LIN {X 0,Y 207.071,Z 348.497,A -85,B 0,C 180,E1 -23061.924,E2 -23061.924} C_VEL
LIN {X 0,Y 208.464,Z 354.265,A -85,B 0,C 180,E1 -23067.075,E2 -23067.075} C_VEL
LIN {X 0,Y 209.704,Z 358.969,A -85,B 0,C 180,E1 -23070.181,E2 -23070.181} C_VEL
LIN {X 0,Y 211.466,Z 367.193,A -85,B 0,C 180,E1 -23074.403,E2 -23074.403} C_VEL
LIN {X 0,Y 212.474,Z 373.609,A -85,B 0,C 180,E1 -23077.134,E2 -23077.134} C_VEL
LIN {X 0,Y 211.976,Z 381.158,A -85,B 0,C 180,E1 -23079.446,E2 -23079.446} C_VEL
LIN {X 0,Y 210.448,Z 390.937,A -85,B 0,C 180,E1 -23082.249,E2 -23082.249} C_VEL
LIN {X 0,Y 208.137,Z 400.366,A -85,B 0,C 180,E1 -23084.841,E2 -23084.841} C_VEL
LIN {X 0,Y 206.322,Z 405.58,A -85,B 0,C 180,E1 -23086.272,E2 -23086.272} C_VEL
LIN {X 0,Y 199.113,Z 417.683,A -85,B 0,C 180,E1 -23089.235,E2 -23089.235} C_VEL
LIN {X 0,Y 192.772,Z 427.559,A -85,B 0,C 180,E1 -23092.364,E2 -23092.364} C_VEL
LIN {X 0,Y 186.872,Z 436.167,A -85,B 0,C 180,E1 -23095.835,E2 -23095.835} C_VEL
LIN {X 0,Y 181.675,Z 443.782,A -85,B 0,C 180,E1 -23099.81,E2 -23099.81} C_VEL
LIN {X 0,Y 177.015,Z 450.226,A -85,B 0,C 180,E1 -23104.106,E2 -23104.106} C_VEL
LIN {X 0,Y 173.093,Z 455.772,A -85,B 0,C 180,E1 -23109.049,E2 -23109.049} C_VEL
LIN {X 0,Y 171.048,Z 459.248,A -85,B 0,C 180,E1 -23113.286,E2 -23113.286} C_VEL
LIN {X 0,Y 169.61,Z 461.995,A -85,B 0,C 180,E1 -23118.045,E2 -23118.045} C_VEL
LIN {X 0,Y 169.147,Z 463.562,A -85,B 0,C 180,E1 -23122.841,E2 -23122.841} C_VEL
LIN {X 0,Y 169.224,Z 463.943,A -85,B 0,C 180,E1 -23125.393,E2 -23125.393} C_VEL
LIN {X 0,Y 169.399,Z 463.779,A -85,B 0,C 180,E1 -23129.986,E2 -23129.986} C_VEL
LIN {X 0,Y 169.181,Z 463.569,A -85,B 0,C 180,E1 -23131.308,E2 -23131.308} C_VEL
LIN {X 0,Y 168.389,Z 463.209,A -85,B 0,C 180,E1 -23132.61,E2 -23132.61} C_VEL
LIN {X 0,Y 165.89,Z 462.118,A -85,B 0,C 180,E1 -23135.171,E2 -23135.171} C_VEL
LIN {X 0,Y 163.361,Z 460.595,A -85,B 0,C 180,E1 -23137.794,E2 -23137.794} C_VEL
LIN {X 0,Y 162.39,Z 459.234,A -85,B 0,C 180,E1 -23139.828,E2 -23139.828} C_VEL
LIN {X 0,Y 162.378,Z 458.73,A -85,B 0,C 180,E1 -23140.514,E2 -23140.514} C_VEL
LIN {X 0,Y 163.318,Z 455.126,A -85,B 0,C 180,E1 -23144.965,E2 -23144.965} C_VEL
LIN {X 0,Y 165.316,Z 449.724,A -85,B 0,C 180,E1 -23149.885,E2 -23149.885} C_VEL
LIN {X 0,Y 168.323,Z 442.8,A -85,B 0,C 180,E1 -23154.68,E2 -23154.68} C_VEL
LIN {X 0,Y 172.5,Z 434.174,A -85,B 0,C 180,E1 -23159.27,E2 -23159.27} C_VEL
LIN {X 0,Y 176.98,Z 424.366,A -85,B 0,C 180,E1 -23163.357,E2 -23163.357} C_VEL
LIN {X 0,Y 182.008,Z 413.854,A -85,B 0,C 180,E1 -23166.765,E2 -23166.765} C_VEL
LIN {X 0,Y 186.944,Z 402.449,A -85,B 0,C 180,E1 -23169.727,E2 -23169.727} C_VEL
LIN {X 0,Y 189.021,Z 397.038,A -85,B 0,C 180,E1 -23170.945,E2 -23170.945} C_VEL
LIN {X 0,Y 189.629,Z 386.332,A -85,B 0,C 180,E1 -23173.653,E2 -23173.653} C_VEL
LIN {X 0,Y 189.573,Z 374.931,A -85,B 0,C 180,E1 -23176.331,E2 -23176.331} C_VEL
LIN {X 0,Y 188.758,Z 362.703,A -85,B 0,C 180,E1 -23179.056,E2 -23179.056} C_VEL
LIN {X 0,Y 187.425,Z 353.021,A -85,B 0,C 180,E1 -23181.158,E2 -23181.158} C_VEL
LIN {X 0,Y 185.608,Z 346.725,A -85,B 0,C 180,E1 -23182.709,E2 -23182.709} C_VEL
LIN {X 0,Y 181.291,Z 336.124,A -85,B 0,C 180,E1 -23185.628,E2 -23185.628} C_VEL
LIN {X 0,Y 177.317,Z 327.465,A -85,B 0,C 180,E1 -23188.151,E2 -23188.151} C_VEL
LIN {X 0,Y 174.427,Z 321.833,A -85,B 0,C 180,E1 -23189.923,E2 -23189.923} C_VEL
LIN {X 0,Y 171.849,Z 316.911,A -85,B 0,C 180,E1 -23191.528,E2 -23191.528} C_VEL
LIN {X 0,Y 169.571,Z 313.23,A -85,B 0,C 180,E1 -23192.874,E2 -23192.874} C_VEL
LIN {X 0,Y 168.653,Z 311.253,A -85,B 0,C 180,E1 -23193.468,E2 -23193.468} C_VEL
LIN {X 0,Y 166.254,Z 308.021,A -85,B 0,C 180,E1 -23194.898,E2 -23194.898} C_VEL
LIN {X 0,Y 165.335,Z 305.195,A -85,B 0,C 180,E1 -23195.68,E2 -23195.68} C_VEL
LIN {X 0,Y 165.069,Z 302.898,A -85,B 0,C 180,E1 -23200.083,E2 -23200.083} C_VEL
LIN {X 0,Y 164.708,Z 300.494,A -85,B 0,C 180,E1 -23205.164,E2 -23205.164} C_VEL
LIN {X 0,Y 164.624,Z 299.609,A -85,B 0,C 180,E1 -23207.673,E2 -23207.673} C_VEL
LIN {X 0,Y 164.832,Z 299.582,A -85,B 0,C 180,E1 -23212.649,E2 -23212.649} C_VEL
LIN {X 0,Y 165.05,Z 299.552,A -85,B 0,C 180,E1 -23217.557,E2 -23217.557} C_VEL
LIN {X 0,Y 165.3,Z 299.52,A -85,B 0,C 180,E1 -23219.997,E2 -23219.997} C_VEL
LIN {X 0,Y 164.865,Z 299.571,A -85,B 0,C 180,E1 -23227.345,E2 -23227.345} C_VEL
LIN {X 0,Y 164.752,Z 299.566,A -85,B 0,C 180,E1 -23231.14,E2 -23231.14} C_VEL
LIN {X 0,Y 164.487,Z 299.615,A -85,B 0,C 180,E1 -23237.4,E2 -23237.4} C_VEL
LIN {X 0,Y 164.476,Z 299.597,A -85,B 0,C 180,E1 -23239.986,E2 -23239.986} C_VEL
LIN {X 0,Y 164.394,Z 299.621,A -85,B 0,C 180,E1 -23246.13,E2 -23246.13} C_VEL
LIN {X 0,Y 164.374,Z 299.633,A -85,B 0,C 180,E1 -23251.224,E2 -23251.224} C_VEL
LIN {X 0,Y 164.311,Z 299.623,A -85,B 0,C 180,E1 -23256.781,E2 -23256.781} C_VEL
LIN {X 0,Y 164.302,Z 299.643,A -85,B 0,C 180,E1 -23259.909,E2 -23259.909} C_VEL
LIN {X 0,Y 164.304,Z 299.623,A -85,B 0,C 180,E1 -23263.349,E2 -23263.349} C_VEL
LIN {X 0,Y 164.354,Z 299.637,A -85,B 0,C 180,E1 -23266.827,E2 -23266.827} C_VEL
LIN {X 0,Y 164.367,Z 299.621,A -85,B 0,C 180,E1 -23270.317,E2 -23270.317} C_VEL
LIN {X 0,Y 164.34,Z 299.626,A -85,B 0,C 180,E1 -23274.339,E2 -23274.339} C_VEL
LIN {X 0,Y 164.38,Z 299.747,A -85,B 0,C 180,E1 -23277.96,E2 -23277.96} C_VEL
LIN {X 0,Y 165.251,Z 302.251,A -85,B 0,C 180,E1 -23278.667,E2 -23278.667} C_VEL
LIN {X 0,Y 167.493,Z 304.644,A -85,B 0,C 180,E1 -23280.056,E2 -23280.056} C_VEL
LIN {X 0,Y 168.139,Z 305.575,A -85,B 0,C 180,E1 -23280.472,E2 -23280.472} C_VEL
LIN {X 0,Y 170.033,Z 308.606,A -85,B 0,C 180,E1 -23281.701,E2 -23281.701} C_VEL
LIN {X 0,Y 171.417,Z 310.257,A -85,B 0,C 180,E1 -23282.532,E2 -23282.532} C_VEL
LIN {X 0,Y 173.819,Z 313.919,A -85,B 0,C 180,E1 -23284.055,E2 -23284.055} C_VEL
LIN {X 0,Y 179.648,Z 323.432,A -85,B 0,C 180,E1 -23287.675,E2 -23287.675} C_VEL
LIN {X 0,Y 184.401,Z 332.346,A -85,B 0,C 180,E1 -23290.779,E2 -23290.779} C_VEL
LIN {X 0,Y 189.654,Z 343.67,A -85,B 0,C 180,E1 -23294.456,E2 -23294.456} C_VEL
LIN {X 0,Y 191.768,Z 349.873,A -85,B 0,C 180,E1 -23296.3,E2 -23296.3} C_VEL
LIN {X 0,Y 193.343,Z 355.545,A -85,B 0,C 180,E1 -23297.935,E2 -23297.935} C_VEL
LIN {X 0,Y 194.691,Z 366.513,A -85,B 0,C 180,E1 -23300.886,E2 -23300.886} C_VEL
LIN {X 0,Y 190.147,Z 378.986,A -85,B 0,C 180,E1 -23303.337,E2 -23303.337} C_VEL
LIN {X 0,Y 185.373,Z 390.665,A -85,B 0,C 180,E1 -23306.194,E2 -23306.194} C_VEL
LIN {X 0,Y 180.718,Z 401.146,A -85,B 0,C 180,E1 -23309.386,E2 -23309.386} C_VEL
LIN {X 0,Y 175.962,Z 411.116,A -85,B 0,C 180,E1 -23313.188,E2 -23313.188} C_VEL
LIN {X 0,Y 172.035,Z 419.15,A -85,B 0,C 180,E1 -23317.038,E2 -23317.038} C_VEL
LIN {X 0,Y 169.033,Z 425.451,A -85,B 0,C 180,E1 -23320.782,E2 -23320.782} C_VEL
LIN {X 0,Y 166.504,Z 430.703,A -85,B 0,C 180,E1 -23324.668,E2 -23324.668} C_VEL
LIN {X 0,Y 164.218,Z 435.982,A -85,B 0,C 180,E1 -23329.7,E2 -23329.7} C_VEL
LIN {X 0,Y 162.694,Z 439.901,A -85,B 0,C 180,E1 -23334.893,E2 -23334.893} C_VEL
LIN {X 0,Y 161.98,Z 442.359,A -85,B 0,C 180,E1 -23339.807,E2 -23339.807} C_VEL
LIN {X 0,Y 161.931,Z 443.673,A -85,B 0,C 180,E1 -23344.456,E2 -23344.456} C_VEL
LIN {X 0,Y 162.435,Z 443.957,A -85,B 0,C 180,E1 -23348.855,E2 -23348.855} C_VEL
LIN {X 0,Y 163.587,Z 443.389,A -85,B 0,C 180,E1 -23353.421,E2 -23353.421} C_VEL
LIN {X 0,Y 165.021,Z 442.215,A -85,B 0,C 180,E1 -23357.05,E2 -23357.05} C_VEL
LIN {X 0,Y 168.232,Z 439.191,A -85,B 0,C 180,E1 -23362.533,E2 -23362.533} C_VEL
LIN {X 0,Y 171.634,Z 435.639,A -85,B 0,C 180,E1 -23366.811,E2 -23366.811} C_VEL
LIN {X 0,Y 176.458,Z 430.293,A -85,B 0,C 180,E1 -23371.452,E2 -23371.452} C_VEL
LIN {X 0,Y 181.905,Z 423.855,A -85,B 0,C 180,E1 -23375.596,E2 -23375.596} C_VEL
LIN {X 0,Y 187.841,Z 416.383,A -85,B 0,C 180,E1 -23379.282,E2 -23379.282} C_VEL
LIN {X 0,Y 194.656,Z 407.022,A -85,B 0,C 180,E1 -23382.818,E2 -23382.818} C_VEL
LIN {X 0,Y 201.597,Z 396.484,A -85,B 0,C 180,E1 -23385.878,E2 -23385.878} C_VEL
LIN {X 0,Y 208.063,Z 385.523,A -85,B 0,C 180,E1 -23388.391,E2 -23388.391} C_VEL
LIN {X 0,Y 209.506,Z 382.789,A -85,B 0,C 180,E1 -23388.942,E2 -23388.942} C_VEL
LIN {X 0,Y 210.087,Z 381.064,A -85,B 0,C 180,E1 -23389.44,E2 -23389.44} C_VEL
LIN {X 0,Y 210.237,Z 375.206,A -85,B 0,C 180,E1 -23391.834,E2 -23391.834} C_VEL
LIN {X 0,Y 209.861,Z 370.028,A -85,B 0,C 180,E1 -23394.236,E2 -23394.236} C_VEL
LIN {X 0,Y 208.905,Z 364.791,A -85,B 0,C 180,E1 -23397.11,E2 -23397.11} C_VEL
LIN {X 0,Y 207.74,Z 360.431,A -85,B 0,C 180,E1 -23400.002,E2 -23400.002} C_VEL
LIN {X 0,Y 206.324,Z 355.745,A -85,B 0,C 180,E1 -23403.908,E2 -23403.908} C_VEL
LIN {X 0,Y 204.735,Z 353.325,A -85,B 0,C 180,E1 -23407.894,E2 -23407.894} C_VEL
LIN {X 0,Y 204.53,Z 351.869,A -85,B 0,C 180,E1 -23409.895,E2 -23409.895} C_VEL
LIN {X 0,Y 203.403,Z 352.092,A -85,B 0,C 180,E1 -23414.663,E2 -23414.663} C_VEL
LIN {X 0,Y 203.38,Z 353.038,A -85,B 0,C 180,E1 -23418.122,E2 -23418.122} C_VEL
LIN {X 0,Y 203.937,Z 354.716,A -85,B 0,C 180,E1 -23421.497,E2 -23421.497} C_VEL
LIN {X 0,Y 205.005,Z 360.752,A -85,B 0,C 180,E1 -23426.962,E2 -23426.962} C_VEL
LIN {X 0,Y 205.992,Z 365.65,A -85,B 0,C 180,E1 -23430.2,E2 -23430.2} C_VEL
LIN {X 0,Y 207.088,Z 372.068,A -85,B 0,C 180,E1 -23433.654,E2 -23433.654} C_VEL
LIN {X 0,Y 207.745,Z 377.925,A -85,B 0,C 180,E1 -23436.302,E2 -23436.302} C_VEL
LIN {X 0,Y 206.849,Z 385.122,A -85,B 0,C 180,E1 -23438.608,E2 -23438.608} C_VEL
LIN {X 0,Y 205.232,Z 393.476,A -85,B 0,C 180,E1 -23441.119,E2 -23441.119} C_VEL
LIN {X 0,Y 202.32,Z 403.303,A -85,B 0,C 180,E1 -23444.009,E2 -23444.009} C_VEL
LIN {X 0,Y 200.971,Z 406.814,A -85,B 0,C 180,E1 -23445.002,E2 -23445.002} C_VEL
LIN {X 0,Y 193.8,Z 418.149,A -85,B 0,C 180,E1 -23447.867,E2 -23447.867} C_VEL
LIN {X 0,Y 187.193,Z 427.848,A -85,B 0,C 180,E1 -23451.036,E2 -23451.036} C_VEL
LIN {X 0,Y 180.722,Z 436.732,A -85,B 0,C 180,E1 -23454.755,E2 -23454.755} C_VEL
LIN {X 0,Y 175.535,Z 443.838,A -85,B 0,C 180,E1 -23458.637,E2 -23458.637} C_VEL
LIN {X 0,Y 170.589,Z 450.155,A -85,B 0,C 180,E1 -23463.054,E2 -23463.054} C_VEL
LIN {X 0,Y 166.237,Z 455.858,A -85,B 0,C 180,E1 -23468.454,E2 -23468.454} C_VEL
LIN {X 0,Y 164.17,Z 458.978,A -85,B 0,C 180,E1 -23472.564,E2 -23472.564} C_VEL
LIN {X 0,Y 162.616,Z 461.65,A -85,B 0,C 180,E1 -23477.522,E2 -23477.522} C_VEL
LIN {X 0,Y 162.069,Z 463.172,A -85,B 0,C 180,E1 -23482.527,E2 -23482.527} C_VEL
LIN {X 0,Y 162.145,Z 463.552,A -85,B 0,C 180,E1 -23485.52,E2 -23485.52} C_VEL
LIN {X 0,Y 162.339,Z 463.282,A -85,B 0,C 180,E1 -23490.002,E2 -23490.002} C_VEL
LIN {X 0,Y 162.26,Z 461.836,A -85,B 0,C 180,E1 -23494.971,E2 -23494.971} C_VEL
LIN {X 0,Y 162.378,Z 458.73,A -85,B 0,C 180,E1 -23500.514,E2 -23500.514} C_VEL
LIN {X 0,Y 162.043,Z 457.229,A -85,B 0,C 180,E1 -23502.525,E2 -23502.525} C_VEL
LIN {X 0,Y 160.054,Z 454.265,A -85,B 0,C 180,E1 -23505.825,E2 -23505.825} C_VEL
LIN {X 0,Y 158.621,Z 451.573,A -85,B 0,C 180,E1 -23508.476,E2 -23508.476} C_VEL
LIN {X 0,Y 158.488,Z 449.287,A -85,B 0,C 180,E1 -23510.456,E2 -23510.456} C_VEL
LIN {X 0,Y 158.733,Z 448.472,A -85,B 0,C 180,E1 -23511.102,E2 -23511.102} C_VEL
LIN {X 0,Y 161.83,Z 441.879,A -85,B 0,C 180,E1 -23515.742,E2 -23515.742} C_VEL
LIN {X 0,Y 165.634,Z 434.34,A -85,B 0,C 180,E1 -23519.907,E2 -23519.907} C_VEL
LIN {X 0,Y 169.816,Z 425.638,A -85,B 0,C 180,E1 -23523.748,E2 -23523.748} C_VEL
LIN {X 0,Y 174.642,Z 415.951,A -85,B 0,C 180,E1 -23527.133,E2 -23527.133} C_VEL
LIN {X 0,Y 179.657,Z 405.016,A -85,B 0,C 180,E1 -23530.202,E2 -23530.202} C_VEL
LIN {X 0,Y 182.279,Z 399.09,A -85,B 0,C 180,E1 -23531.591,E2 -23531.591} C_VEL
LIN {X 0,Y 183.038,Z 393.259,A -85,B 0,C 180,E1 -23533.15,E2 -23533.15} C_VEL
LIN {X 0,Y 183.591,Z 381.901,A -85,B 0,C 180,E1 -23536.063,E2 -23536.063} C_VEL
LIN {X 0,Y 183.191,Z 368.545,A -85,B 0,C 180,E1 -23539.29,E2 -23539.29} C_VEL
LIN {X 0,Y 182.089,Z 357.305,A -85,B 0,C 180,E1 -23541.861,E2 -23541.861} C_VEL
LIN {X 0,Y 180.742,Z 351.699,A -85,B 0,C 180,E1 -23543.293,E2 -23543.293} C_VEL
LIN {X 0,Y 177.021,Z 341.596,A -85,B 0,C 180,E1 -23546.23,E2 -23546.23} C_VEL
LIN {X 0,Y 172.562,Z 331.508,A -85,B 0,C 180,E1 -23549.394,E2 -23549.394} C_VEL
LIN {X 0,Y 170.204,Z 326.59,A -85,B 0,C 180,E1 -23551.016,E2 -23551.016} C_VEL
LIN {X 0,Y 167.936,Z 322.038,A -85,B 0,C 180,E1 -23552.588,E2 -23552.588} C_VEL
LIN {X 0,Y 165.635,Z 317.842,A -85,B 0,C 180,E1 -23554.133,E2 -23554.133} C_VEL
LIN {X 0,Y 164.649,Z 316.146,A -85,B 0,C 180,E1 -23554.814,E2 -23554.814} C_VEL
LIN {X 0,Y 162.454,Z 312.456,A -85,B 0,C 180,E1 -23556.324,E2 -23556.324} C_VEL
LIN {X 0,Y 161.827,Z 310.898,A -85,B 0,C 180,E1 -23556.82,E2 -23556.82} C_VEL
LIN {X 0,Y 159.384,Z 307.951,A -85,B 0,C 180,E1 -23558.451,E2 -23558.451} C_VEL
LIN {X 0,Y 158.244,Z 305.128,A -85,B 0,C 180,E1 -23559.392,E2 -23559.392} C_VEL
LIN {X 0,Y 158.127,Z 304.535,A -85,B 0,C 180,E1 -23559.613,E2 -23559.613} C_VEL
LIN {X 0,Y 157.788,Z 302.272,A -85,B 0,C 180,E1 -23564.497,E2 -23564.497} C_VEL
LIN {X 0,Y 157.664,Z 300.477,A -85,B 0,C 180,E1 -23568.724,E2 -23568.724} C_VEL
LIN {X 0,Y 157.77,Z 300.461,A -85,B 0,C 180,E1 -23572.318,E2 -23572.318} C_VEL
LIN {X 0,Y 158.262,Z 300.396,A -85,B 0,C 180,E1 -23579.997,E2 -23579.997} C_VEL
LIN {X 0,Y 157.824,Z 300.449,A -85,B 0,C 180,E1 -23587.674,E2 -23587.674} C_VEL
LIN {X 0,Y 157.681,Z 300.445,A -85,B 0,C 180,E1 -23591.308,E2 -23591.308} C_VEL
LIN {X 0,Y 157.458,Z 300.494,A -85,B 0,C 180,E1 -23595.531,E2 -23595.531} C_VEL
LIN {X 0,Y 157.372,Z 300.482,A -85,B 0,C 180,E1 -23600.929,E2 -23600.929} C_VEL
LIN {X 0,Y 157.314,Z 300.496,A -85,B 0,C 180,E1 -23606.68,E2 -23606.68} C_VEL
LIN {X 0,Y 157.276,Z 300.519,A -85,B 0,C 180,E1 -23612.424,E2 -23612.424} C_VEL
LIN {X 0,Y 157.28,Z 300.496,A -85,B 0,C 180,E1 -23616.452,E2 -23616.452} C_VEL
LIN {X 0,Y 157.23,Z 300.505,A -85,B 0,C 180,E1 -23622.1,E2 -23622.1} C_VEL
LIN {X 0,Y 157.267,Z 300.508,A -85,B 0,C 180,E1 -23627.906,E2 -23627.906} C_VEL
LIN {X 0,Y 157.318,Z 300.506,A -85,B 0,C 180,E1 -23633.521,E2 -23633.521} C_VEL
LIN {X 0,Y 157.344,Z 300.741,A -85,B 0,C 180,E1 -23634.173,E2 -23634.173} C_VEL
LIN {X 0,Y 158.263,Z 303.328,A -85,B 0,C 180,E1 -23635.031,E2 -23635.031} C_VEL
LIN {X 0,Y 160.468,Z 305.585,A -85,B 0,C 180,E1 -23636.597,E2 -23636.597} C_VEL
LIN {X 0,Y 161.163,Z 306.274,A -85,B 0,C 180,E1 -23637.078,E2 -23637.078} C_VEL
LIN {X 0,Y 162.882,Z 309.263,A -85,B 0,C 180,E1 -23638.399,E2 -23638.399} C_VEL
LIN {X 0,Y 164.628,Z 311.207,A -85,B 0,C 180,E1 -23639.561,E2 -23639.561} C_VEL
LIN {X 0,Y 166.622,Z 314.493,A -85,B 0,C 180,E1 -23641.01,E2 -23641.01} C_VEL
LIN {X 0,Y 167.879,Z 316.234,A -85,B 0,C 180,E1 -23641.835,E2 -23641.835} C_VEL
LIN {X 0,Y 171.316,Z 321.865,A -85,B 0,C 180,E1 -23644.257,E2 -23644.257} C_VEL
LIN {X 0,Y 176.674,Z 331.015,A -85,B 0,C 180,E1 -23647.907,E2 -23647.907} C_VEL
LIN {X 0,Y 182.095,Z 342.603,A -85,B 0,C 180,E1 -23652.014,E2 -23652.014} C_VEL
LIN {X 0,Y 185.244,Z 350.27,A -85,B 0,C 180,E1 -23654.597,E2 -23654.597} C_VEL
LIN {X 0,Y 187.458,Z 358.394,A -85,B 0,C 180,E1 -23657.089,E2 -23657.089} C_VEL
LIN {X 0,Y 188.504,Z 368.436,A -85,B 0,C 180,E1 -23659.928,E2 -23659.928} C_VEL
LIN {X 0,Y 183.632,Z 380.952,A -85,B 0,C 180,E1 -23662.488,E2 -23662.488} C_VEL
LIN {X 0,Y 178.599,Z 392.604,A -85,B 0,C 180,E1 -23665.485,E2 -23665.485} C_VEL
LIN {X 0,Y 173.762,Z 402.994,A -85,B 0,C 180,E1 -23668.84,E2 -23668.84} C_VEL
LIN {X 0,Y 168.862,Z 412.738,A -85,B 0,C 180,E1 -23672.783,E2 -23672.783} C_VEL
LIN {X 0,Y 164.93,Z 420.448,A -85,B 0,C 180,E1 -23676.728,E2 -23676.728} C_VEL
LIN {X 0,Y 161.385,Z 427.521,A -85,B 0,C 180,E1 -23681.299,E2 -23681.299} C_VEL
LIN {X 0,Y 158.962,Z 432.55,A -85,B 0,C 180,E1 -23685.381,E2 -23685.381} C_VEL
LIN {X 0,Y 156.975,Z 436.866,A -85,B 0,C 180,E1 -23689.925,E2 -23689.925} C_VEL
LIN {X 0,Y 155.485,Z 440.626,A -85,B 0,C 180,E1 -23695.318,E2 -23695.318} C_VEL
LIN {X 0,Y 154.848,Z 442.958,A -85,B 0,C 180,E1 -23700.426,E2 -23700.426} C_VEL
LIN {X 0,Y 154.965,Z 444.269,A -85,B 0,C 180,E1 -23706.125,E2 -23706.125} C_VEL
LIN {X 0,Y 155.498,Z 444.413,A -85,B 0,C 180,E1 -23709.8,E2 -23709.8} C_VEL
LIN {X 0,Y 157.283,Z 443.484,A -85,B 0,C 180,E1 -23715.636,E2 -23715.636} C_VEL
LIN {X 0,Y 158.728,Z 442.37,A -85,B 0,C 180,E1 -23718.823,E2 -23718.823} C_VEL
LIN {X 0,Y 160.797,Z 440.621,A -85,B 0,C 180,E1 -23722.277,E2 -23722.277} C_VEL
LIN {X 0,Y 163.682,Z 437.907,A -85,B 0,C 180,E1 -23726.074,E2 -23726.074} C_VEL
LIN {X 0,Y 168.555,Z 432.978,A -85,B 0,C 180,E1 -23731.113,E2 -23731.113} C_VEL
LIN {X 0,Y 173.661,Z 427.534,A -85,B 0,C 180,E1 -23735.193,E2 -23735.193} C_VEL
LIN {X 0,Y 180.165,Z 420.023,A -85,B 0,C 180,E1 -23739.419,E2 -23739.419} C_VEL
LIN {X 0,Y 186.354,Z 412.349,A -85,B 0,C 180,E1 -23742.718,E2 -23742.718} C_VEL
LIN {X 0,Y 192.976,Z 403.363,A -85,B 0,C 180,E1 -23745.767,E2 -23745.767} C_VEL
LIN {X 0,Y 199.726,Z 393.198,A -85,B 0,C 180,E1 -23748.458,E2 -23748.458} C_VEL
LIN {X 0,Y 204.156,Z 385.756,A -85,B 0,C 180,E1 -23750.091,E2 -23750.091} C_VEL
LIN {X 0,Y 204.883,Z 383.863,A -85,B 0,C 180,E1 -23750.625,E2 -23750.625} C_VEL
LIN {X 0,Y 205.216,Z 379.272,A -85,B 0,C 180,E1 -23752.649,E2 -23752.649} C_VEL
LIN {X 0,Y 205.061,Z 374.382,A -85,B 0,C 180,E1 -23755.087,E2 -23755.087} C_VEL
LIN {X 0,Y 204.429,Z 369.435,A -85,B 0,C 180,E1 -23758.032,E2 -23758.032} C_VEL
LIN {X 0,Y 203.564,Z 365.487,A -85,B 0,C 180,E1 -23760.892,E2 -23760.892} C_VEL
LIN {X 0,Y 202.715,Z 361.961,A -85,B 0,C 180,E1 -23763.978,E2 -23763.978} C_VEL
LIN {X 0,Y 201.203,Z 358.172,A -85,B 0,C 180,E1 -23770.06,E2 -23770.06} C_VEL
LIN {X 0,Y 200.253,Z 358.359,A -85,B 0,C 180,E1 -23774.223,E2 -23774.223} C_VEL
LIN {X 0,Y 200.183,Z 359.594,A -85,B 0,C 180,E1 -23778.579,E2 -23778.579} C_VEL
LIN {X 0,Y 200.468,Z 360.511,A -85,B 0,C 180,E1 -23780.525,E2 -23780.525} C_VEL
LIN {X 0,Y 201.162,Z 365.751,A -85,B 0,C 180,E1 -23785.896,E2 -23785.896} C_VEL
LIN {X 0,Y 201.924,Z 370.937,A -85,B 0,C 180,E1 -23789.529,E2 -23789.529} C_VEL
LIN {X 0,Y 202.642,Z 377.1,A -85,B 0,C 180,E1 -23793.029,E2 -23793.029} C_VEL
LIN {X 0,Y 202.955,Z 381.759,A -85,B 0,C 180,E1 -23795.278,E2 -23795.278} C_VEL
LIN {X 0,Y 202.051,Z 387.505,A -85,B 0,C 180,E1 -23797.255,E2 -23797.255} C_VEL
LIN {X 0,Y 200.052,Z 395.773,A -85,B 0,C 180,E1 -23799.896,E2 -23799.896} C_VEL
LIN {X 0,Y 197.106,Z 404.716,A -85,B 0,C 180,E1 -23802.648,E2 -23802.648} C_VEL
LIN {X 0,Y 195.828,Z 407.785,A -85,B 0,C 180,E1 -23803.6,E2 -23803.6} C_VEL
LIN {X 0,Y 188.608,Z 418.614,A -85,B 0,C 180,E1 -23806.423,E2 -23806.423} C_VEL
LIN {X 0,Y 181.727,Z 428.159,A -85,B 0,C 180,E1 -23809.628,E2 -23809.628} C_VEL
LIN {X 0,Y 175.476,Z 436.238,A -85,B 0,C 180,E1 -23813.077,E2 -23813.077} C_VEL
LIN {X 0,Y 169.445,Z 443.886,A -85,B 0,C 180,E1 -23817.373,E2 -23817.373} C_VEL
LIN {X 0,Y 164.216,Z 450.105,A -85,B 0,C 180,E1 -23821.918,E2 -23821.918} C_VEL
LIN {X 0,Y 160.148,Z 455.007,A -85,B 0,C 180,E1 -23826.739,E2 -23826.739} C_VEL
LIN {X 0,Y 157.32,Z 458.716,A -85,B 0,C 180,E1 -23831.779,E2 -23831.779} C_VEL
LIN {X 0,Y 155.625,Z 461.3,A -85,B 0,C 180,E1 -23836.952,E2 -23836.952} C_VEL
LIN {X 0,Y 154.983,Z 462.779,A -85,B 0,C 180,E1 -23842.183,E2 -23842.183} C_VEL
LIN {X 0,Y 155.068,Z 463.107,A -85,B 0,C 180,E1 -23845.65,E2 -23845.65} C_VEL
LIN {X 0,Y 155.277,Z 462.781,A -85,B 0,C 180,E1 -23850.002,E2 -23850.002} C_VEL
LIN {X 0,Y 155.172,Z 461.256,A -85,B 0,C 180,E1 -23855.199,E2 -23855.199} C_VEL
LIN {X 0,Y 155.293,Z 458.348,A -85,B 0,C 180,E1 -23860.592,E2 -23860.592} C_VEL
LIN {X 0,Y 156.403,Z 454.383,A -85,B 0,C 180,E1 -23865.643,E2 -23865.643} C_VEL
LIN {X 0,Y 158.564,Z 448.902,A -85,B 0,C 180,E1 -23870.77,E2 -23870.77} C_VEL
LIN {X 0,Y 158.733,Z 448.472,A -85,B 0,C 180,E1 -23871.102,E2 -23871.102} C_VEL
LIN {X 0,Y 159.159,Z 446.011,A -85,B 0,C 180,E1 -23873.019,E2 -23873.019} C_VEL
LIN {X 0,Y 158.148,Z 437.709,A -85,B 0,C 180,E1 -23878.723,E2 -23878.723} C_VEL
LIN {X 0,Y 158.829,Z 434.554,A -85,B 0,C 180,E1 -23880.527,E2 -23880.527} C_VEL
LIN {X 0,Y 159.338,Z 433.472,A -85,B 0,C 180,E1 -23881.095,E2 -23881.095} C_VEL
LIN {X 0,Y 164.278,Z 423.629,A -85,B 0,C 180,E1 -23885.483,E2 -23885.483} C_VEL
LIN {X 0,Y 169.824,Z 412.941,A -85,B 0,C 180,E1 -23889.134,E2 -23889.134} C_VEL
LIN {X 0,Y 175.16,Z 401.523,A -85,B 0,C 180,E1 -23892.229,E2 -23892.229} C_VEL
LIN {X 0,Y 176.078,Z 399.372,A -85,B 0,C 180,E1 -23892.732,E2 -23892.732} C_VEL
LIN {X 0,Y 177.005,Z 390.945,A -85,B 0,C 180,E1 -23895.123,E2 -23895.123} C_VEL
LIN {X 0,Y 177.472,Z 380.203,A -85,B 0,C 180,E1 -23897.963,E2 -23897.963} C_VEL
LIN {X 0,Y 177.194,Z 368.166,A -85,B 0,C 180,E1 -23900.974,E2 -23900.974} C_VEL
LIN {X 0,Y 176.3,Z 358.771,A -85,B 0,C 180,E1 -23903.274,E2 -23903.274} C_VEL
LIN {X 0,Y 173.995,Z 351.045,A -85,B 0,C 180,E1 -23905.561,E2 -23905.561} C_VEL
LIN {X 0,Y 170.017,Z 340.659,A -85,B 0,C 180,E1 -23908.885,E2 -23908.885} C_VEL
LIN {X 0,Y 166.188,Z 331.804,A -85,B 0,C 180,E1 -23911.933,E2 -23911.933} C_VEL
LIN {X 0,Y 163.798,Z 326.918,A -85,B 0,C 180,E1 -23913.736,E2 -23913.736} C_VEL
LIN {X 0,Y 161.266,Z 321.824,A -85,B 0,C 180,E1 -23915.733,E2 -23915.733} C_VEL
LIN {X 0,Y 159.052,Z 317.877,A -85,B 0,C 180,E1 -23917.424,E2 -23917.424} C_VEL
LIN {X 0,Y 158.142,Z 316.204,A -85,B 0,C 180,E1 -23918.146,E2 -23918.146} C_VEL
LIN {X 0,Y 155.74,Z 312.547,A -85,B 0,C 180,E1 -23920.002,E2 -23920.002} C_VEL
LIN {X 0,Y 154.818,Z 310.335,A -85,B 0,C 180,E1 -23920.834,E2 -23920.834} C_VEL
LIN {X 0,Y 152.167,Z 307.28,A -85,B 0,C 180,E1 -23922.96,E2 -23922.96} C_VEL
LIN {X 0,Y 150.98,Z 304.414,A -85,B 0,C 180,E1 -23924.126,E2 -23924.126} C_VEL
LIN {X 0,Y 150.854,Z 303.71,A -85,B 0,C 180,E1 -23924.459,E2 -23924.459} C_VEL
LIN {X 0,Y 150.705,Z 301.743,A -85,B 0,C 180,E1 -23929.247,E2 -23929.247} C_VEL
LIN {X 0,Y 150.708,Z 301.341,A -85,B 0,C 180,E1 -23931.955,E2 -23931.955} C_VEL
LIN {X 0,Y 151.223,Z 301.273,A -85,B 0,C 180,E1 -23939.997,E2 -23939.997} C_VEL
LIN {X 0,Y 150.76,Z 301.33,A -85,B 0,C 180,E1 -23948.036,E2 -23948.036} C_VEL
LIN {X 0,Y 150.617,Z 301.323,A -85,B 0,C 180,E1 -23951.501,E2 -23951.501} C_VEL
LIN {X 0,Y 150.366,Z 301.379,A -85,B 0,C 180,E1 -23956.283,E2 -23956.283} C_VEL
LIN {X 0,Y 150.353,Z 301.355,A -85,B 0,C 180,E1 -23960.789,E2 -23960.789} C_VEL
LIN {X 0,Y 150.244,Z 301.371,A -85,B 0,C 180,E1 -23967.278,E2 -23967.278} C_VEL
LIN {X 0,Y 150.216,Z 301.397,A -85,B 0,C 180,E1 -23972.63,E2 -23972.63} C_VEL
LIN {X 0,Y 150.21,Z 301.383,A -85,B 0,C 180,E1 -23977.458,E2 -23977.458} C_VEL
LIN {X 0,Y 150.167,Z 301.387,A -85,B 0,C 180,E1 -23981.509,E2 -23981.509} C_VEL
LIN {X 0,Y 150.191,Z 301.398,A -85,B 0,C 180,E1 -23985.417,E2 -23985.417} C_VEL
LIN {X 0,Y 150.243,Z 301.443,A -85,B 0,C 180,E1 -23989.541,E2 -23989.541} C_VEL
LIN {X 0,Y 151.047,Z 303.92,A -85,B 0,C 180,E1 -23990.465,E2 -23990.465} C_VEL
LIN {X 0,Y 153.156,Z 306.295,A -85,B 0,C 180,E1 -23992.328,E2 -23992.328} C_VEL
LIN {X 0,Y 154.312,Z 307.206,A -85,B 0,C 180,E1 -23993.23,E2 -23993.23} C_VEL
LIN {X 0,Y 155.813,Z 310.107,A -85,B 0,C 180,E1 -23994.612,E2 -23994.612} C_VEL
LIN {X 0,Y 157.98,Z 312.384,A -85,B 0,C 180,E1 -23996.248,E2 -23996.248} C_VEL
LIN {X 0,Y 160.126,Z 315.829,A -85,B 0,C 180,E1 -23998.022,E2 -23998.022} C_VEL
LIN {X 0,Y 161.25,Z 317.342,A -85,B 0,C 180,E1 -23998.86,E2 -23998.86} C_VEL
LIN {X 0,Y 164.585,Z 322.714,A -85,B 0,C 180,E1 -24001.463,E2 -24001.463} C_VEL
LIN {X 0,Y 167.702,Z 328.055,A -85,B 0,C 180,E1 -24003.868,E2 -24003.868} C_VEL
LIN {X 0,Y 172.436,Z 336.848,A -85,B 0,C 180,E1 -24007.518,E2 -24007.518} C_VEL
LIN {X 0,Y 177.12,Z 347.429,A -85,B 0,C 180,E1 -24011.491,E2 -24011.491} C_VEL
LIN {X 0,Y 179.944,Z 354.869,A -85,B 0,C 180,E1 -24014.132,E2 -24014.132} C_VEL
LIN {X 0,Y 181.709,Z 362.448,A -85,B 0,C 180,E1 -24016.58,E2 -24016.58} C_VEL
LIN {X 0,Y 182.286,Z 370.245,A -85,B 0,C 180,E1 -24018.884,E2 -24018.884} C_VEL
LIN {X 0,Y 177.354,Z 382.363,A -85,B 0,C 180,E1 -24021.471,E2 -24021.471} C_VEL
LIN {X 0,Y 171.906,Z 394.437,A -85,B 0,C 180,E1 -24024.72,E2 -24024.72} C_VEL
LIN {X 0,Y 166.901,Z 404.617,A -85,B 0,C 180,E1 -24028.189,E2 -24028.189} C_VEL
LIN {X 0,Y 161.602,Z 414.626,A -85,B 0,C 180,E1 -24032.491,E2 -24032.491} C_VEL
LIN {X 0,Y 157.281,Z 422.816,A -85,B 0,C 180,E1 -24037.057,E2 -24037.057} C_VEL
LIN {X 0,Y 153.725,Z 429.543,A -85,B 0,C 180,E1 -24041.87,E2 -24041.87} C_VEL
LIN {X 0,Y 150.76,Z 435.635,A -85,B 0,C 180,E1 -24047.637,E2 -24047.637} C_VEL
LIN {X 0,Y 149.159,Z 439.139,A -85,B 0,C 180,E1 -24052.142,E2 -24052.142} C_VEL
LIN {X 0,Y 148.295,Z 441.355,A -85,B 0,C 180,E1 -24055.791,E2 -24055.791} C_VEL
LIN {X 0,Y 147.695,Z 443.711,A -85,B 0,C 180,E1 -24061.56,E2 -24061.56} C_VEL
LIN {X 0,Y 147.894,Z 444.676,A -85,B 0,C 180,E1 -24066.12,E2 -24066.12} C_VEL
LIN {X 0,Y 148.759,Z 444.86,A -85,B 0,C 180,E1 -24071.405,E2 -24071.405} C_VEL
LIN {X 0,Y 150.013,Z 444.261,A -85,B 0,C 180,E1 -24075.358,E2 -24075.358} C_VEL
LIN {X 0,Y 152.966,Z 442.194,A -85,B 0,C 180,E1 -24081.355,E2 -24081.355} C_VEL
LIN {X 0,Y 156.396,Z 439.398,A -85,B 0,C 180,E1 -24086.146,E2 -24086.146} C_VEL
LIN {X 0,Y 161.36,Z 434.871,A -85,B 0,C 180,E1 -24091.377,E2 -24091.377} C_VEL
LIN {X 0,Y 166.742,Z 429.572,A -85,B 0,C 180,E1 -24095.736,E2 -24095.736} C_VEL
LIN {X 0,Y 172.502,Z 423.462,A -85,B 0,C 180,E1 -24099.557,E2 -24099.557} C_VEL
LIN {X 0,Y 179.633,Z 415.327,A -85,B 0,C 180,E1 -24103.438,E2 -24103.438} C_VEL
LIN {X 0,Y 186.109,Z 407.2,A -85,B 0,C 180,E1 -24106.442,E2 -24106.442} C_VEL
LIN {X 0,Y 193.14,Z 397.488,A -85,B 0,C 180,E1 -24109.25,E2 -24109.25} C_VEL
LIN {X 0,Y 199.034,Z 388.427,A -85,B 0,C 180,E1 -24111.366,E2 -24111.366} C_VEL
LIN {X 0,Y 199.831,Z 386.613,A -85,B 0,C 180,E1 -24111.915,E2 -24111.915} C_VEL
LIN {X 0,Y 200.28,Z 382.337,A -85,B 0,C 180,E1 -24113.959,E2 -24113.959} C_VEL
LIN {X 0,Y 200.155,Z 377.05,A -85,B 0,C 180,E1 -24116.983,E2 -24116.983} C_VEL
LIN {X 0,Y 199.668,Z 372.626,A -85,B 0,C 180,E1 -24120.002,E2 -24120.002} C_VEL
LIN {X 0,Y 198.87,Z 368.033,A -85,B 0,C 180,E1 -24124.055,E2 -24124.055} C_VEL
LIN {X 0,Y 197.641,Z 364.34,A -85,B 0,C 180,E1 -24130.244,E2 -24130.244} C_VEL
LIN {X 0,Y 196.704,Z 364.793,A -85,B 0,C 180,E1 -24135.28,E2 -24135.28} C_VEL
LIN {X 0,Y 196.715,Z 365.907,A -85,B 0,C 180,E1 -24138.758,E2 -24138.758} C_VEL
LIN {X 0,Y 196.877,Z 367.18,A -85,B 0,C 180,E1 -24140.917,E2 -24140.917} C_VEL
LIN {X 0,Y 197.28,Z 371.347,A -85,B 0,C 180,E1 -24145.311,E2 -24145.311} C_VEL
LIN {X 0,Y 197.686,Z 375.828,A -85,B 0,C 180,E1 -24148.684,E2 -24148.684} C_VEL
LIN {X 0,Y 198.102,Z 383.05,A -85,B 0,C 180,E1 -24152.941,E2 -24152.941} C_VEL
LIN {X 0,Y 198.035,Z 386.466,A -85,B 0,C 180,E1 -24154.6,E2 -24154.6} C_VEL
LIN {X 0,Y 196.672,Z 392.411,A -85,B 0,C 180,E1 -24156.687,E2 -24156.687} C_VEL
LIN {X 0,Y 194.326,Z 399.979,A -85,B 0,C 180,E1 -24159.228,E2 -24159.228} C_VEL
LIN {X 0,Y 191.232,Z 407.83,A -85,B 0,C 180,E1 -24161.788,E2 -24161.788} C_VEL
LIN {X 0,Y 190.256,Z 409.781,A -85,B 0,C 180,E1 -24162.374,E2 -24162.374} C_VEL
LIN {X 0,Y 183.545,Z 419.15,A -85,B 0,C 180,E1 -24164.9,E2 -24164.9} C_VEL
LIN {X 0,Y 176.377,Z 428.481,A -85,B 0,C 180,E1 -24168.133,E2 -24168.133} C_VEL
LIN {X 0,Y 169.834,Z 436.412,A -85,B 0,C 180,E1 -24171.633,E2 -24171.633} C_VEL
LIN {X 0,Y 163.454,Z 443.942,A -85,B 0,C 180,E1 -24176.018,E2 -24176.018} C_VEL
LIN {X 0,Y 157.931,Z 450.055,A -85,B 0,C 180,E1 -24180.694,E2 -24180.694} C_VEL
LIN {X 0,Y 153.579,Z 454.858,A -85,B 0,C 180,E1 -24185.681,E2 -24185.681} C_VEL
LIN {X 0,Y 150.503,Z 458.47,A -85,B 0,C 180,E1 -24190.923,E2 -24190.923} C_VEL
LIN {X 0,Y 148.638,Z 460.957,A -85,B 0,C 180,E1 -24196.327,E2 -24196.327} C_VEL
LIN {X 0,Y 147.924,Z 462.359,A -85,B 0,C 180,E1 -24201.808,E2 -24201.808} C_VEL
LIN {X 0,Y 148.005,Z 462.637,A -85,B 0,C 180,E1 -24205.727,E2 -24205.727} C_VEL
LIN {X 0,Y 148.216,Z 462.279,A -85,B 0,C 180,E1 -24210.002,E2 -24210.002} C_VEL
LIN {X 0,Y 148.066,Z 460.666,A -85,B 0,C 180,E1 -24215.449,E2 -24215.449} C_VEL
LIN {X 0,Y 148.25,Z 457.785,A -85,B 0,C 180,E1 -24220.933,E2 -24220.933} C_VEL
LIN {X 0,Y 149.521,Z 453.615,A -85,B 0,C 180,E1 -24226.383,E2 -24226.383} C_VEL
LIN {X 0,Y 151.838,Z 448.031,A -85,B 0,C 180,E1 -24231.735,E2 -24231.735} C_VEL
LIN {X 0,Y 155.349,Z 440.902,A -85,B 0,C 180,E1 -24236.9,E2 -24236.9} C_VEL
LIN {X 0,Y 159.338,Z 433.472,A -85,B 0,C 180,E1 -24241.095,E2 -24241.095} C_VEL
LIN {X 0,Y 160.49,Z 430.154,A -85,B 0,C 180,E1 -24242.795,E2 -24242.795} C_VEL
LIN {X 0,Y 160.823,Z 424.386,A -85,B 0,C 180,E1 -24245.669,E2 -24245.669} C_VEL
LIN {X 0,Y 161.407,Z 418.26,A -85,B 0,C 180,E1 -24248.426,E2 -24248.426} C_VEL
LIN {X 0,Y 162.907,Z 414.257,A -85,B 0,C 180,E1 -24249.883,E2 -24249.883} C_VEL
LIN {X 0,Y 167.944,Z 404.049,A -85,B 0,C 180,E1 -24252.847,E2 -24252.847} C_VEL
LIN {X 0,Y 169.833,Z 399.938,A -85,B 0,C 180,E1 -24253.882,E2 -24253.882} C_VEL
LIN {X 0,Y 171.132,Z 388.294,A -85,B 0,C 180,E1 -24257.293,E2 -24257.293} C_VEL
LIN {X 0,Y 171.522,Z 376.29,A -85,B 0,C 180,E1 -24260.571,E2 -24260.571} C_VEL
LIN {X 0,Y 171.037,Z 363.905,A -85,B 0,C 180,E1 -24263.792,E2 -24263.792} C_VEL
LIN {X 0,Y 170.149,Z 359.328,A -85,B 0,C 180,E1 -24265.116,E2 -24265.116} C_VEL
LIN {X 0,Y 167.047,Z 349.72,A -85,B 0,C 180,E1 -24268.269,E2 -24268.269} C_VEL
LIN {X 0,Y 162.676,Z 338.282,A -85,B 0,C 180,E1 -24272.324,E2 -24272.324} C_VEL
LIN {X 0,Y 159.817,Z 332.002,A -85,B 0,C 180,E1 -24274.783,E2 -24274.783} C_VEL
LIN {X 0,Y 157.287,Z 326.777,A -85,B 0,C 180,E1 -24276.982,E2 -24276.982} C_VEL
LIN {X 0,Y 154.771,Z 321.804,A -85,B 0,C 180,E1 -24279.219,E2 -24279.219} C_VEL
LIN {X 0,Y 152.359,Z 317.661,A -85,B 0,C 180,E1 -24281.334,E2 -24281.334} C_VEL
LIN {X 0,Y 151.58,Z 316.028,A -85,B 0,C 180,E1 -24282.109,E2 -24282.109} C_VEL
LIN {X 0,Y 149.089,Z 312.559,A -85,B 0,C 180,E1 -24284.358,E2 -24284.358} C_VEL
LIN {X 0,Y 147.804,Z 309.719,A -85,B 0,C 180,E1 -24285.717,E2 -24285.717} C_VEL
LIN {X 0,Y 145.271,Z 306.776,A -85,B 0,C 180,E1 -24288.243,E2 -24288.243} C_VEL
LIN {X 0,Y 143.813,Z 303.453,A -85,B 0,C 180,E1 -24290.06,E2 -24290.06} C_VEL
LIN {X 0,Y 143.685,Z 302.857,A -85,B 0,C 180,E1 -24290.318,E2 -24290.318} C_VEL
LIN {X 0,Y 143.681,Z 302.4,A -85,B 0,C 180,E1 -24291.559,E2 -24291.559} C_VEL
LIN {X 0,Y 144.181,Z 302.15,A -85,B 0,C 180,E1 -24299.997,E2 -24299.997} C_VEL
LIN {X 0,Y 143.678,Z 302.212,A -85,B 0,C 180,E1 -24308.435,E2 -24308.435} C_VEL
LIN {X 0,Y 143.552,Z 302.201,A -85,B 0,C 180,E1 -24311.709,E2 -24311.709} C_VEL
LIN {X 0,Y 143.305,Z 302.254,A -85,B 0,C 180,E1 -24317.109,E2 -24317.109} C_VEL
LIN {X 0,Y 143.279,Z 302.237,A -85,B 0,C 180,E1 -24321.251,E2 -24321.251} C_VEL
LIN {X 0,Y 143.19,Z 302.247,A -85,B 0,C 180,E1 -24327.933,E2 -24327.933} C_VEL
LIN {X 0,Y 143.166,Z 302.267,A -85,B 0,C 180,E1 -24333.43,E2 -24333.43} C_VEL
LIN {X 0,Y 143.08,Z 302.287,A -85,B 0,C 180,E1 -24339.679,E2 -24339.679} C_VEL
LIN {X 0,Y 143.105,Z 302.414,A -85,B 0,C 180,E1 -24343.698,E2 -24343.698} C_VEL
LIN {X 0,Y 144.055,Z 304.962,A -85,B 0,C 180,E1 -24345.031,E2 -24345.031} C_VEL
LIN {X 0,Y 146.083,Z 307.204,A -85,B 0,C 180,E1 -24347.29,E2 -24347.29} C_VEL
LIN {X 0,Y 147.43,Z 308.01,A -85,B 0,C 180,E1 -24348.533,E2 -24348.533} C_VEL
LIN {X 0,Y 148.88,Z 310.943,A -85,B 0,C 180,E1 -24350.16,E2 -24350.16} C_VEL
LIN {X 0,Y 151.388,Z 313.633,A -85,B 0,C 180,E1 -24352.454,E2 -24352.454} C_VEL
LIN {X 0,Y 153.154,Z 316.681,A -85,B 0,C 180,E1 -24354.199,E2 -24354.199} C_VEL
LIN {X 0,Y 154.774,Z 318.544,A -85,B 0,C 180,E1 -24355.529,E2 -24355.529} C_VEL
LIN {X 0,Y 156.986,Z 322.036,A -85,B 0,C 180,E1 -24357.503,E2 -24357.503} C_VEL
LIN {X 0,Y 162.342,Z 331.055,A -85,B 0,C 180,E1 -24362.098,E2 -24362.098} C_VEL
LIN {X 0,Y 167.364,Z 340.927,A -85,B 0,C 180,E1 -24366.486,E2 -24366.486} C_VEL
LIN {X 0,Y 171.543,Z 350.823,A -85,B 0,C 180,E1 -24370.431,E2 -24370.431} C_VEL
LIN {X 0,Y 174.544,Z 359.297,A -85,B 0,C 180,E1 -24373.628,E2 -24373.628} C_VEL
LIN {X 0,Y 175.853,Z 365.505,A -85,B 0,C 180,E1 -24375.744,E2 -24375.744} C_VEL
LIN {X 0,Y 176.168,Z 371.986,A -85,B 0,C 180,E1 -24377.768,E2 -24377.768} C_VEL
LIN {X 0,Y 170.863,Z 384.363,A -85,B 0,C 180,E1 -24380.528,E2 -24380.528} C_VEL
LIN {X 0,Y 165.221,Z 396.207,A -85,B 0,C 180,E1 -24383.894,E2 -24383.894} C_VEL
LIN {X 0,Y 160.038,Z 406.217,A -85,B 0,C 180,E1 -24387.481,E2 -24387.481} C_VEL
LIN {X 0,Y 154.687,Z 415.796,A -85,B 0,C 180,E1 -24391.845,E2 -24391.845} C_VEL
LIN {X 0,Y 150.167,Z 423.997,A -85,B 0,C 180,E1 -24396.702,E2 -24396.702} C_VEL
LIN {X 0,Y 146.998,Z 429.745,A -85,B 0,C 180,E1 -24401.023,E2 -24401.023} C_VEL
LIN {X 0,Y 144.485,Z 434.519,A -85,B 0,C 180,E1 -24405.55,E2 -24405.55} C_VEL
LIN {X 0,Y 142.543,Z 438.601,A -85,B 0,C 180,E1 -24410.492,E2 -24410.492} C_VEL
LIN {X 0,Y 141.028,Z 442.214,A -85,B 0,C 180,E1 -24416.646,E2 -24416.646} C_VEL
LIN {X 0,Y 140.594,Z 444.142,A -85,B 0,C 180,E1 -24421.818,E2 -24421.818} C_VEL
LIN {X 0,Y 140.882,Z 445.169,A -85,B 0,C 180,E1 -24427.05,E2 -24427.05} C_VEL
LIN {X 0,Y 141.805,Z 445.328,A -85,B 0,C 180,E1 -24431.982,E2 -24431.982} C_VEL
LIN {X 0,Y 143.61,Z 444.526,A -85,B 0,C 180,E1 -24437.226,E2 -24437.226} C_VEL
LIN {X 0,Y 145.594,Z 443.313,A -85,B 0,C 180,E1 -24441.137,E2 -24441.137} C_VEL
LIN {X 0,Y 150.098,Z 439.995,A -85,B 0,C 180,E1 -24447.434,E2 -24447.434} C_VEL
LIN {X 0,Y 155.856,Z 435.134,A -85,B 0,C 180,E1 -24453.2,E2 -24453.2} C_VEL
LIN {X 0,Y 162.633,Z 428.892,A -85,B 0,C 180,E1 -24458.29,E2 -24458.29} C_VEL
LIN {X 0,Y 169.528,Z 421.918,A -85,B 0,C 180,E1 -24462.452,E2 -24462.452} C_VEL
LIN {X 0,Y 177.166,Z 413.418,A -85,B 0,C 180,E1 -24466.233,E2 -24466.233} C_VEL
LIN {X 0,Y 184.381,Z 404.587,A -85,B 0,C 180,E1 -24469.248,E2 -24469.248} C_VEL
LIN {X 0,Y 191.658,Z 394.584,A -85,B 0,C 180,E1 -24471.909,E2 -24471.909} C_VEL
LIN {X 0,Y 194.524,Z 390.219,A -85,B 0,C 180,E1 -24472.905,E2 -24472.905} C_VEL
LIN {X 0,Y 195.22,Z 386.355,A -85,B 0,C 180,E1 -24474.839,E2 -24474.839} C_VEL
LIN {X 0,Y 195.368,Z 381.337,A -85,B 0,C 180,E1 -24477.941,E2 -24477.941} C_VEL
LIN {X 0,Y 195.171,Z 377.262,A -85,B 0,C 180,E1 -24481.034,E2 -24481.034} C_VEL
LIN {X 0,Y 194.786,Z 373.968,A -85,B 0,C 180,E1 -24484.14,E2 -24484.14} C_VEL
LIN {X 0,Y 193.911,Z 371.55,A -85,B 0,C 180,E1 -24488.338,E2 -24488.338} C_VEL
LIN {X 0,Y 193.848,Z 370.371,A -85,B 0,C 180,E1 -24490.446,E2 -24490.446} C_VEL
LIN {X 0,Y 193.056,Z 370.749,A -85,B 0,C 180,E1 -24494.765,E2 -24494.765} C_VEL
LIN {X 0,Y 192.986,Z 372.218,A -85,B 0,C 180,E1 -24499.135,E2 -24499.135} C_VEL
LIN {X 0,Y 192.98,Z 374.59,A -85,B 0,C 180,E1 -24502.316,E2 -24502.316} C_VEL
LIN {X 0,Y 193.192,Z 376.69,A -85,B 0,C 180,E1 -24504.574,E2 -24504.574} C_VEL
LIN {X 0,Y 193.311,Z 381.237,A -85,B 0,C 180,E1 -24508.207,E2 -24508.207} C_VEL
LIN {X 0,Y 193.321,Z 388.017,A -85,B 0,C 180,E1 -24512.406,E2 -24512.406} C_VEL
LIN {X 0,Y 192.965,Z 391.253,A -85,B 0,C 180,E1 -24513.958,E2 -24513.958} C_VEL
LIN {X 0,Y 189.997,Z 400.302,A -85,B 0,C 180,E1 -24517.235,E2 -24517.235} C_VEL
LIN {X 0,Y 186.2,Z 409.174,A -85,B 0,C 180,E1 -24520.289,E2 -24520.289} C_VEL
LIN {X 0,Y 184.402,Z 412.113,A -85,B 0,C 180,E1 -24521.176,E2 -24521.176} C_VEL
LIN {X 0,Y 177.535,Z 421.149,A -85,B 0,C 180,E1 -24523.745,E2 -24523.745} C_VEL
LIN {X 0,Y 170.121,Z 430.092,A -85,B 0,C 180,E1 -24527.03,E2 -24527.03} C_VEL
LIN {X 0,Y 162.576,Z 438.515,A -85,B 0,C 180,E1 -24531.092,E2 -24531.092} C_VEL
LIN {X 0,Y 156.018,Z 445.628,A -85,B 0,C 180,E1 -24535.734,E2 -24535.734} C_VEL
LIN {X 0,Y 150.448,Z 451.271,A -85,B 0,C 180,E1 -24540.629,E2 -24540.629} C_VEL
LIN {X 0,Y 145.726,Z 456.048,A -85,B 0,C 180,E1 -24546.4,E2 -24546.4} C_VEL
LIN {X 0,Y 142.552,Z 459.56,A -85,B 0,C 180,E1 -24552.796,E2 -24552.796} C_VEL
LIN {X 0,Y 141.137,Z 461.411,A -85,B 0,C 180,E1 -24558.513,E2 -24558.513} C_VEL
LIN {X 0,Y 140.849,Z 462.182,A -85,B 0,C 180,E1 -24564.275,E2 -24564.275} C_VEL
LIN {X 0,Y 140.949,Z 462.139,A -85,B 0,C 180,E1 -24567.144,E2 -24567.144} C_VEL
LIN {X 0,Y 141.132,Z 461.774,A -85,B 0,C 180,E1 -24570.002,E2 -24570.002} C_VEL
LIN {X 0,Y 141.025,Z 460.501,A -85,B 0,C 180,E1 -24574.624,E2 -24574.624} C_VEL
LIN {X 0,Y 140.96,Z 458.75,A -85,B 0,C 180,E1 -24578.604,E2 -24578.604} C_VEL
LIN {X 0,Y 141.831,Z 455.151,A -85,B 0,C 180,E1 -24584.347,E2 -24584.347} C_VEL
LIN {X 0,Y 143.76,Z 450.19,A -85,B 0,C 180,E1 -24590.013,E2 -24590.013} C_VEL
LIN {X 0,Y 146.944,Z 443.756,A -85,B 0,C 180,E1 -24595.498,E2 -24595.498} C_VEL
LIN {X 0,Y 151.331,Z 435.672,A -85,B 0,C 180,E1 -24600.723,E2 -24600.723} C_VEL
LIN {X 0,Y 156.044,Z 427.032,A -85,B 0,C 180,E1 -24605.049,E2 -24605.049} C_VEL
LIN {X 0,Y 160.783,Z 418.281,A -85,B 0,C 180,E1 -24608.529,E2 -24608.529} C_VEL
LIN {X 0,Y 162.907,Z 414.257,A -85,B 0,C 180,E1 -24609.883,E2 -24609.883} C_VEL
LIN {X 0,Y 164.409,Z 410.167,A -85,B 0,C 180,E1 -24611.29,E2 -24611.29} C_VEL
LIN {X 0,Y 164.902,Z 406.057,A -85,B 0,C 180,E1 -24612.787,E2 -24612.787} C_VEL
LIN {X 0,Y 164.582,Z 397.716,A -85,B 0,C 180,E1 -24615.855,E2 -24615.855} C_VEL
LIN {X 0,Y 164.761,Z 391.807,A -85,B 0,C 180,E1 -24617.799,E2 -24617.799} C_VEL
LIN {X 0,Y 165.485,Z 381.706,A -85,B 0,C 180,E1 -24620.783,E2 -24620.783} C_VEL
LIN {X 0,Y 165.563,Z 370.965,A -85,B 0,C 180,E1 -24623.761,E2 -24623.761} C_VEL
LIN {X 0,Y 165.275,Z 365.324,A -85,B 0,C 180,E1 -24625.316,E2 -24625.316} C_VEL
LIN {X 0,Y 163.095,Z 357.033,A -85,B 0,C 180,E1 -24628.136,E2 -24628.136} C_VEL
LIN {X 0,Y 159.281,Z 345.922,A -85,B 0,C 180,E1 -24632.255,E2 -24632.255} C_VEL
LIN {X 0,Y 156.246,Z 337.948,A -85,B 0,C 180,E1 -24635.411,E2 -24635.411} C_VEL
LIN {X 0,Y 153.218,Z 331.569,A -85,B 0,C 180,E1 -24638.293,E2 -24638.293} C_VEL
LIN {X 0,Y 151.228,Z 327.32,A -85,B 0,C 180,E1 -24640.307,E2 -24640.307} C_VEL
LIN {X 0,Y 148.939,Z 322.731,A -85,B 0,C 180,E1 -24642.69,E2 -24642.69} C_VEL
LIN {X 0,Y 145.843,Z 317.604,A -85,B 0,C 180,E1 -24645.871,E2 -24645.871} C_VEL
LIN {X 0,Y 145.012,Z 315.748,A -85,B 0,C 180,E1 -24646.891,E2 -24646.891} C_VEL
LIN {X 0,Y 142.563,Z 312.3,A -85,B 0,C 180,E1 -24649.701,E2 -24649.701} C_VEL
LIN {X 0,Y 141.184,Z 309.111,A -85,B 0,C 180,E1 -24651.589,E2 -24651.589} C_VEL
LIN {X 0,Y 138.298,Z 306.898,A -85,B 0,C 180,E1 -24655.26,E2 -24655.26} C_VEL
LIN {X 0,Y 137.146,Z 304.561,A -85,B 0,C 180,E1 -24657.243,E2 -24657.243} C_VEL
LIN {X 0,Y 136.873,Z 303.061,A -85,B 0,C 180,E1 -24658.066,E2 -24658.066} C_VEL
LIN {X 0,Y 137.138,Z 303.027,A -85,B 0,C 180,E1 -24659.997,E2 -24659.997} C_VEL
LIN {X 0,Y 136.603,Z 303.091,A -85,B 0,C 180,E1 -24668.876,E2 -24668.876} C_VEL
LIN {X 0,Y 136.495,Z 303.078,A -85,B 0,C 180,E1 -24671.951,E2 -24671.951} C_VEL
LIN {X 0,Y 136.245,Z 303.121,A -85,B 0,C 180,E1 -24678.026,E2 -24678.026} C_VEL
LIN {X 0,Y 136.2,Z 303.121,A -85,B 0,C 180,E1 -24681.745,E2 -24681.745} C_VEL
LIN {X 0,Y 136.1,Z 303.129,A -85,B 0,C 180,E1 -24688.612,E2 -24688.612} C_VEL
LIN {X 0,Y 136.058,Z 303.137,A -85,B 0,C 180,E1 -24695.298,E2 -24695.298} C_VEL
LIN {X 0,Y 136.3,Z 304.193,A -85,B 0,C 180,E1 -24696.135,E2 -24696.135} C_VEL
LIN {X 0,Y 137.3,Z 306.365,A -85,B 0,C 180,E1 -24698.052,E2 -24698.052} C_VEL
LIN {X 0,Y 139.675,Z 308.507,A -85,B 0,C 180,E1 -24701.525,E2 -24701.525} C_VEL
LIN {X 0,Y 140.741,Z 309.246,A -85,B 0,C 180,E1 -24702.836,E2 -24702.836} C_VEL
LIN {X 0,Y 142.291,Z 312.252,A -85,B 0,C 180,E1 -24705.01,E2 -24705.01} C_VEL
LIN {X 0,Y 144.782,Z 314.676,A -85,B 0,C 180,E1 -24707.818,E2 -24707.818} C_VEL
LIN {X 0,Y 146.561,Z 317.812,A -85,B 0,C 180,E1 -24709.937,E2 -24709.937} C_VEL
LIN {X 0,Y 148.274,Z 319.732,A -85,B 0,C 180,E1 -24711.592,E2 -24711.592} C_VEL
LIN {X 0,Y 150.477,Z 323.347,A -85,B 0,C 180,E1 -24713.962,E2 -24713.962} C_VEL
LIN {X 0,Y 151.348,Z 324.548,A -85,B 0,C 180,E1 -24714.785,E2 -24714.785} C_VEL
LIN {X 0,Y 156.509,Z 333.348,A -85,B 0,C 180,E1 -24719.781,E2 -24719.781} C_VEL
LIN {X 0,Y 161.688,Z 343.633,A -85,B 0,C 180,E1 -24724.806,E2 -24724.806} C_VEL
LIN {X 0,Y 165.649,Z 353.303,A -85,B 0,C 180,E1 -24728.962,E2 -24728.962} C_VEL
LIN {X 0,Y 168.681,Z 362.008,A -85,B 0,C 180,E1 -24732.528,E2 -24732.528} C_VEL
LIN {X 0,Y 169.98,Z 369.464,A -85,B 0,C 180,E1 -24735.218,E2 -24735.218} C_VEL
LIN {X 0,Y 170.062,Z 373.624,A -85,B 0,C 180,E1 -24736.577,E2 -24736.577} C_VEL
LIN {X 0,Y 164.784,Z 385.413,A -85,B 0,C 180,E1 -24739.301,E2 -24739.301} C_VEL
LIN {X 0,Y 159.487,Z 396.122,A -85,B 0,C 180,E1 -24742.402,E2 -24742.402} C_VEL
LIN {X 0,Y 153.911,Z 406.467,A -85,B 0,C 180,E1 -24746.186,E2 -24746.186} C_VEL
LIN {X 0,Y 148.309,Z 416.053,A -85,B 0,C 180,E1 -24750.671,E2 -24750.671} C_VEL
LIN {X 0,Y 143.633,Z 424.151,A -85,B 0,C 180,E1 -24755.614,E2 -24755.614} C_VEL
LIN {X 0,Y 140.274,Z 429.914,A -85,B 0,C 180,E1 -24760.097,E2 -24760.097} C_VEL
LIN {X 0,Y 136.912,Z 436.133,A -85,B 0,C 180,E1 -24766.397,E2 -24766.397} C_VEL
LIN {X 0,Y 135.115,Z 439.734,A -85,B 0,C 180,E1 -24771.35,E2 -24771.35} C_VEL
LIN {X 0,Y 133.9,Z 442.709,A -85,B 0,C 180,E1 -24776.848,E2 -24776.848} C_VEL
LIN {X 0,Y 133.513,Z 444.731,A -85,B 0,C 180,E1 -24782.632,E2 -24782.632} C_VEL
LIN {X 0,Y 134.031,Z 445.749,A -85,B 0,C 180,E1 -24788.99,E2 -24788.99} C_VEL
LIN {X 0,Y 135.007,Z 445.786,A -85,B 0,C 180,E1 -24793.22,E2 -24793.22} C_VEL
LIN {X 0,Y 137.708,Z 444.641,A -85,B 0,C 180,E1 -24799.951,E2 -24799.951} C_VEL
LIN {X 0,Y 139.8,Z 443.377,A -85,B 0,C 180,E1 -24803.544,E2 -24803.544} C_VEL
LIN {X 0,Y 143.832,Z 440.631,A -85,B 0,C 180,E1 -24808.763,E2 -24808.763} C_VEL
LIN {X 0,Y 148.852,Z 436.75,A -85,B 0,C 180,E1 -24813.772,E2 -24813.772} C_VEL
LIN {X 0,Y 155.467,Z 431.211,A -85,B 0,C 180,E1 -24818.802,E2 -24818.802} C_VEL
LIN {X 0,Y 163.093,Z 424.128,A -85,B 0,C 180,E1 -24823.431,E2 -24823.431} C_VEL
LIN {X 0,Y 171.075,Z 415.963,A -85,B 0,C 180,E1 -24827.33,E2 -24827.33} C_VEL
LIN {X 0,Y 178.238,Z 407.804,A -85,B 0,C 180,E1 -24830.309,E2 -24830.309} C_VEL
LIN {X 0,Y 186.521,Z 397.276,A -85,B 0,C 180,E1 -24833.256,E2 -24833.256} C_VEL
LIN {X 0,Y 189.175,Z 393.619,A -85,B 0,C 180,E1 -24834.139,E2 -24834.139} C_VEL
LIN {X 0,Y 189.818,Z 392.172,A -85,B 0,C 180,E1 -24834.691,E2 -24834.691} C_VEL
LIN {X 0,Y 190.381,Z 388.645,A -85,B 0,C 180,E1 -24836.827,E2 -24836.827} C_VEL
LIN {X 0,Y 190.61,Z 384.243,A -85,B 0,C 180,E1 -24840.002,E2 -24840.002} C_VEL
LIN {X 0,Y 190.498,Z 380.742,A -85,B 0,C 180,E1 -24843.175,E2 -24843.175} C_VEL
LIN {X 0,Y 190.424,Z 379.291,A -85,B 0,C 180,E1 -24844.82,E2 -24844.82} C_VEL
LIN {X 0,Y 189.841,Z 376.273,A -85,B 0,C 180,E1 -24850.669,E2 -24850.669} C_VEL
LIN {X 0,Y 189.097,Z 376.773,A -85,B 0,C 180,E1 -24855.082,E2 -24855.082} C_VEL
LIN {X 0,Y 189.007,Z 377.395,A -85,B 0,C 180,E1 -24857.308,E2 -24857.308} C_VEL
LIN {X 0,Y 188.95,Z 378.486,A -85,B 0,C 180,E1 -24859.56,E2 -24859.56} C_VEL
LIN {X 0,Y 188.847,Z 381.17,A -85,B 0,C 180,E1 -24863.004,E2 -24863.004} C_VEL
LIN {X 0,Y 188.863,Z 383.387,A -85,B 0,C 180,E1 -24865.176,E2 -24865.176} C_VEL
LIN {X 0,Y 188.77,Z 386.503,A -85,B 0,C 180,E1 -24867.736,E2 -24867.736} C_VEL
LIN {X 0,Y 188.443,Z 392.205,A -85,B 0,C 180,E1 -24871.477,E2 -24871.477} C_VEL
LIN {X 0,Y 188.066,Z 394.61,A -85,B 0,C 180,E1 -24872.749,E2 -24872.749} C_VEL
LIN {X 0,Y 185.687,Z 401.063,A -85,B 0,C 180,E1 -24875.254,E2 -24875.254} C_VEL
LIN {X 0,Y 182.128,Z 408.935,A -85,B 0,C 180,E1 -24878.13,E2 -24878.13} C_VEL
LIN {X 0,Y 179.825,Z 412.878,A -85,B 0,C 180,E1 -24879.48,E2 -24879.48} C_VEL
LIN {X 0,Y 171.574,Z 422.998,A -85,B 0,C 180,E1 -24882.5,E2 -24882.5} C_VEL
LIN {X 0,Y 162.892,Z 432.672,A -85,B 0,C 180,E1 -24886.347,E2 -24886.347} C_VEL
LIN {X 0,Y 155.16,Z 440.661,A -85,B 0,C 180,E1 -24890.647,E2 -24890.647} C_VEL
LIN {X 0,Y 148.541,Z 447.174,A -85,B 0,C 180,E1 -24895.408,E2 -24895.408} C_VEL
LIN {X 0,Y 142.981,Z 452.396,A -85,B 0,C 180,E1 -24900.561,E2 -24900.561} C_VEL
LIN {X 0,Y 138.608,Z 456.436,A -85,B 0,C 180,E1 -24906.071,E2 -24906.071} C_VEL
LIN {X 0,Y 135.709,Z 459.279,A -85,B 0,C 180,E1 -24911.899,E2 -24911.899} C_VEL
LIN {X 0,Y 134.134,Z 461.03,A -85,B 0,C 180,E1 -24917.904,E2 -24917.904} C_VEL
LIN {X 0,Y 133.747,Z 461.71,A -85,B 0,C 180,E1 -24923.97,E2 -24923.97} C_VEL
LIN {X 0,Y 133.879,Z 461.635,A -85,B 0,C 180,E1 -24926.993,E2 -24926.993} C_VEL
LIN {X 0,Y 134.05,Z 461.257,A -85,B 0,C 180,E1 -24930.002,E2 -24930.002} C_VEL
LIN {X 0,Y 133.936,Z 460.056,A -85,B 0,C 180,E1 -24934.421,E2 -24934.421} C_VEL
LIN {X 0,Y 133.91,Z 458.096,A -85,B 0,C 180,E1 -24939.061,E2 -24939.061} C_VEL
LIN {X 0,Y 134.883,Z 454.396,A -85,B 0,C 180,E1 -24945.103,E2 -24945.103} C_VEL
LIN {X 0,Y 137.029,Z 449.332,A -85,B 0,C 180,E1 -24951.042,E2 -24951.042} C_VEL
LIN {X 0,Y 140.473,Z 442.784,A -85,B 0,C 180,E1 -24956.764,E2 -24956.764} C_VEL
LIN {X 0,Y 145.207,Z 434.581,A -85,B 0,C 180,E1 -24962.17,E2 -24962.17} C_VEL
LIN {X 0,Y 150.163,Z 425.79,A -85,B 0,C 180,E1 -24966.638,E2 -24966.638} C_VEL
LIN {X 0,Y 156.108,Z 415.249,A -85,B 0,C 180,E1 -24970.755,E2 -24970.755} C_VEL
LIN {X 0,Y 161.733,Z 404.428,A -85,B 0,C 180,E1 -24974.051,E2 -24974.051} C_VEL
LIN {X 0,Y 163.633,Z 400.377,A -85,B 0,C 180,E1 -24975.129,E2 -24975.129} C_VEL
LIN {X 0,Y 164.761,Z 391.807,A -85,B 0,C 180,E1 -24977.799,E2 -24977.799} C_VEL
LIN {X 0,Y 164.808,Z 388.969,A -85,B 0,C 180,E1 -24978.73,E2 -24978.73} C_VEL
LIN {X 0,Y 163.998,Z 384.928,A -85,B 0,C 180,E1 -24980.228,E2 -24980.228} C_VEL
LIN {X 0,Y 160.737,Z 376.092,A -85,B 0,C 180,E1 -24983.89,E2 -24983.89} C_VEL
LIN {X 0,Y 159.912,Z 371.888,A -85,B 0,C 180,E1 -24985.388,E2 -24985.388} C_VEL
LIN {X 0,Y 159.833,Z 370.366,A -85,B 0,C 180,E1 -24985.85,E2 -24985.85} C_VEL
LIN {X 0,Y 159.285,Z 366.273,A -85,B 0,C 180,E1 -24987.205,E2 -24987.205} C_VEL
LIN {X 0,Y 156.89,Z 357.527,A -85,B 0,C 180,E1 -24990.476,E2 -24990.476} C_VEL
LIN {X 0,Y 153.31,Z 346.549,A -85,B 0,C 180,E1 -24994.908,E2 -24994.908} C_VEL
LIN {X 0,Y 150.266,Z 338.74,A -85,B 0,C 180,E1 -24998.385,E2 -24998.385} C_VEL
LIN {X 0,Y 147.483,Z 332.518,A -85,B 0,C 180,E1 -25001.549,E2 -25001.549} C_VEL
LIN {X 0,Y 145.065,Z 327.454,A -85,B 0,C 180,E1 -25004.375,E2 -25004.375} C_VEL
LIN {X 0,Y 142.775,Z 323.149,A -85,B 0,C 180,E1 -25007.143,E2 -25007.143} C_VEL
LIN {X 0,Y 142.116,Z 321.702,A -85,B 0,C 180,E1 -25008.063,E2 -25008.063} C_VEL
LIN {X 0,Y 139.733,Z 317.809,A -85,B 0,C 180,E1 -25011.136,E2 -25011.136} C_VEL
LIN {X 0,Y 138.87,Z 315.615,A -85,B 0,C 180,E1 -25012.546,E2 -25012.546} C_VEL
LIN {X 0,Y 136.202,Z 313.243,A -85,B 0,C 180,E1 -25016.299,E2 -25016.299} C_VEL
LIN {X 0,Y 135.082,Z 310.573,A -85,B 0,C 180,E1 -25018.599,E2 -25018.599} C_VEL
LIN {X 0,Y 134.797,Z 309.762,A -85,B 0,C 180,E1 -25019.25,E2 -25019.25} C_VEL
LIN {X 0,Y 130.963,Z 307.457,A -85,B 0,C 180,E1 -25028.095,E2 -25028.095} C_VEL
LIN {X 0,Y 130.1,Z 306.282,A -85,B 0,C 180,E1 -25032.475,E2 -25032.475} C_VEL
LIN {X 0,Y 129.781,Z 306.114,A -85,B 0,C 180,E1 -25038.957,E2 -25038.957} C_VEL
LIN {X 0,Y 130.034,Z 306.727,A -85,B 0,C 180,E1 -25042.227,E2 -25042.227} C_VEL
LIN {X 0,Y 133.541,Z 309.768,A -85,B 0,C 180,E1 -25053.595,E2 -25053.595} C_VEL
LIN {X 0,Y 134.123,Z 310.113,A -85,B 0,C 180,E1 -25054.717,E2 -25054.717} C_VEL
LIN {X 0,Y 135.16,Z 312.814,A -85,B 0,C 180,E1 -25057.186,E2 -25057.186} C_VEL
LIN {X 0,Y 137.336,Z 315.054,A -85,B 0,C 180,E1 -25060.706,E2 -25060.706} C_VEL
LIN {X 0,Y 138.317,Z 315.859,A -85,B 0,C 180,E1 -25062.073,E2 -25062.073} C_VEL
LIN {X 0,Y 140.09,Z 319.108,A -85,B 0,C 180,E1 -25064.795,E2 -25064.795} C_VEL
LIN {X 0,Y 141.953,Z 320.999,A -85,B 0,C 180,E1 -25067.033,E2 -25067.033} C_VEL
LIN {X 0,Y 143.864,Z 324.357,A -85,B 0,C 180,E1 -25069.566,E2 -25069.566} C_VEL
LIN {X 0,Y 145.092,Z 325.956,A -85,B 0,C 180,E1 -25070.909,E2 -25070.909} C_VEL
LIN {X 0,Y 149.202,Z 332.901,A -85,B 0,C 180,E1 -25075.578,E2 -25075.578} C_VEL
LIN {X 0,Y 152.97,Z 339.897,A -85,B 0,C 180,E1 -25079.641,E2 -25079.641} C_VEL
LIN {X 0,Y 157.441,Z 349.651,A -85,B 0,C 180,E1 -25084.605,E2 -25084.605} C_VEL
LIN {X 0,Y 160.842,Z 358.813,A -85,B 0,C 180,E1 -25088.761,E2 -25088.761} C_VEL
LIN {X 0,Y 163.184,Z 366.146,A -85,B 0,C 180,E1 -25091.914,E2 -25091.914} C_VEL
LIN {X 0,Y 164.093,Z 372.19,A -85,B 0,C 180,E1 -25094.24,E2 -25094.24} C_VEL
LIN {X 0,Y 164.109,Z 374.622,A -85,B 0,C 180,E1 -25095.109,E2 -25095.109} C_VEL
LIN {X 0,Y 162.164,Z 379.365,A -85,B 0,C 180,E1 -25096.208,E2 -25096.208} C_VEL
LIN {X 0,Y 156.379,Z 391.142,A -85,B 0,C 180,E1 -25099.283,E2 -25099.283} C_VEL
LIN {X 0,Y 150.941,Z 401.289,A -85,B 0,C 180,E1 -25102.642,E2 -25102.642} C_VEL
LIN {X 0,Y 145.506,Z 410.624,A -85,B 0,C 180,E1 -25106.537,E2 -25106.537} C_VEL
LIN {X 0,Y 140.564,Z 418.673,A -85,B 0,C 180,E1 -25110.779,E2 -25110.779} C_VEL
LIN {X 0,Y 135.918,Z 426.291,A -85,B 0,C 180,E1 -25115.934,E2 -25115.934} C_VEL
LIN {X 0,Y 132.544,Z 431.826,A -85,B 0,C 180,E1 -25120.693,E2 -25120.693} C_VEL
LIN {X 0,Y 129.289,Z 437.676,A -85,B 0,C 180,E1 -25127.394,E2 -25127.394} C_VEL
LIN {X 0,Y 127.587,Z 441.087,A -85,B 0,C 180,E1 -25132.678,E2 -25132.678} C_VEL
LIN {X 0,Y 126.707,Z 443.342,A -85,B 0,C 180,E1 -25137.452,E2 -25137.452} C_VEL
LIN {X 0,Y 126.442,Z 445.354,A -85,B 0,C 180,E1 -25143.765,E2 -25143.765} C_VEL
LIN {X 0,Y 126.981,Z 446.157,A -85,B 0,C 180,E1 -25149.215,E2 -25149.215} C_VEL
LIN {X 0,Y 128.518,Z 446.147,A -85,B 0,C 180,E1 -25155.305,E2 -25155.305} C_VEL
LIN {X 0,Y 130.347,Z 445.475,A -85,B 0,C 180,E1 -25159.688,E2 -25159.688} C_VEL
LIN {X 0,Y 133.122,Z 444.098,A -85,B 0,C 180,E1 -25164.502,E2 -25164.502} C_VEL
LIN {X 0,Y 137.647,Z 441.287,A -85,B 0,C 180,E1 -25170.221,E2 -25170.221} C_VEL
LIN {X 0,Y 143.025,Z 437.487,A -85,B 0,C 180,E1 -25175.37,E2 -25175.37} C_VEL
LIN {X 0,Y 150.713,Z 431.503,A -85,B 0,C 180,E1 -25180.952,E2 -25180.952} C_VEL
LIN {X 0,Y 157.742,Z 425.4,A -85,B 0,C 180,E1 -25185.029,E2 -25185.029} C_VEL
LIN {X 0,Y 166.398,Z 417.075,A -85,B 0,C 180,E1 -25189.1,E2 -25189.1} C_VEL
LIN {X 0,Y 173.841,Z 409.109,A -85,B 0,C 180,E1 -25192.073,E2 -25192.073} C_VEL
LIN {X 0,Y 181.726,Z 399.741,A -85,B 0,C 180,E1 -25194.755,E2 -25194.755} C_VEL
LIN {X 0,Y 184.381,Z 396.21,A -85,B 0,C 180,E1 -25195.63,E2 -25195.63} C_VEL
LIN {X 0,Y 185.09,Z 394.14,A -85,B 0,C 180,E1 -25196.773,E2 -25196.773} C_VEL
LIN {X 0,Y 185.728,Z 389.805,A -85,B 0,C 180,E1 -25200.002,E2 -25200.002} C_VEL
LIN {X 0,Y 185.88,Z 387.336,A -85,B 0,C 180,E1 -25202.169,E2 -25202.169} C_VEL
LIN {X 0,Y 185.978,Z 385.338,A -85,B 0,C 180,E1 -25204.337,E2 -25204.337} C_VEL
LIN {X 0,Y 185.791,Z 383.913,A -85,B 0,C 180,E1 -25206.518,E2 -25206.518} C_VEL
LIN {X 0,Y 185.6,Z 382.048,A -85,B 0,C 180,E1 -25210.916,E2 -25210.916} C_VEL
LIN {X 0,Y 184.907,Z 382.657,A -85,B 0,C 180,E1 -25215.432,E2 -25215.432} C_VEL
LIN {X 0,Y 184.758,Z 383.514,A -85,B 0,C 180,E1 -25218.021,E2 -25218.021} C_VEL
LIN {X 0,Y 184.644,Z 384.637,A -85,B 0,C 180,E1 -25220.035,E2 -25220.035} C_VEL
LIN {X 0,Y 184.442,Z 387.727,A -85,B 0,C 180,E1 -25223.869,E2 -25223.869} C_VEL
LIN {X 0,Y 184.048,Z 391.65,A -85,B 0,C 180,E1 -25227.275,E2 -25227.275} C_VEL
LIN {X 0,Y 183.414,Z 397.026,A -85,B 0,C 180,E1 -25230.956,E2 -25230.956} C_VEL
LIN {X 0,Y 182.664,Z 399.422,A -85,B 0,C 180,E1 -25232.175,E2 -25232.175} C_VEL
LIN {X 0,Y 178.904,Z 407.507,A -85,B 0,C 180,E1 -25235.368,E2 -25235.368} C_VEL
LIN {X 0,Y 175.374,Z 413.652,A -85,B 0,C 180,E1 -25237.68,E2 -25237.68} C_VEL
LIN {X 0,Y 166.873,Z 423.563,A -85,B 0,C 180,E1 -25240.707,E2 -25240.707} C_VEL
LIN {X 0,Y 157.821,Z 433.043,A -85,B 0,C 180,E1 -25244.564,E2 -25244.564} C_VEL
LIN {X 0,Y 149.707,Z 440.836,A -85,B 0,C 180,E1 -25248.914,E2 -25248.914} C_VEL
LIN {X 0,Y 142.723,Z 447.215,A -85,B 0,C 180,E1 -25253.781,E2 -25253.781} C_VEL
LIN {X 0,Y 136.791,Z 452.305,A -85,B 0,C 180,E1 -25259.087,E2 -25259.087} C_VEL
LIN {X 0,Y 132.083,Z 456.216,A -85,B 0,C 180,E1 -25264.809,E2 -25264.809} C_VEL
LIN {X 0,Y 128.91,Z 459.007,A -85,B 0,C 180,E1 -25270.909,E2 -25270.909} C_VEL
LIN {X 0,Y 127.139,Z 460.655,A -85,B 0,C 180,E1 -25277.228,E2 -25277.228} C_VEL
LIN {X 0,Y 126.653,Z 461.239,A -85,B 0,C 180,E1 -25283.63,E2 -25283.63} C_VEL
LIN {X 0,Y 126.793,Z 461.121,A -85,B 0,C 180,E1 -25286.825,E2 -25286.825} C_VEL
LIN {X 0,Y 126.969,Z 460.706,A -85,B 0,C 180,E1 -25290.002,E2 -25290.002} C_VEL
LIN {X 0,Y 126.853,Z 459.605,A -85,B 0,C 180,E1 -25294.216,E2 -25294.216} C_VEL
LIN {X 0,Y 126.864,Z 457.443,A -85,B 0,C 180,E1 -25299.569,E2 -25299.569} C_VEL
LIN {X 0,Y 127.971,Z 453.642,A -85,B 0,C 180,E1 -25305.94,E2 -25305.94} C_VEL
LIN {X 0,Y 130.346,Z 448.472,A -85,B 0,C 180,E1 -25312.176,E2 -25312.176} C_VEL
LIN {X 0,Y 134.086,Z 441.811,A -85,B 0,C 180,E1 -25318.149,E2 -25318.149} C_VEL
LIN {X 0,Y 138.467,Z 434.617,A -85,B 0,C 180,E1 -25323.07,E2 -25323.07} C_VEL
LIN {X 0,Y 143.628,Z 425.927,A -85,B 0,C 180,E1 -25327.711,E2 -25327.711} C_VEL
LIN {X 0,Y 148.864,Z 417.14,A -85,B 0,C 180,E1 -25331.375,E2 -25331.375} C_VEL
LIN {X 0,Y 154.619,Z 406.776,A -85,B 0,C 180,E1 -25334.794,E2 -25334.794} C_VEL
LIN {X 0,Y 157.46,Z 401.065,A -85,B 0,C 180,E1 -25336.394,E2 -25336.394} C_VEL
LIN {X 0,Y 159.044,Z 389.917,A -85,B 0,C 180,E1 -25340.01,E2 -25340.01} C_VEL
LIN {X 0,Y 159.833,Z 377.114,A -85,B 0,C 180,E1 -25343.873,E2 -25343.873} C_VEL
LIN {X 0,Y 159.833,Z 370.366,A -85,B 0,C 180,E1 -25345.85,E2 -25345.85} C_VEL
LIN {X 0,Y 159.432,Z 367.56,A -85,B 0,C 180,E1 -25346.806,E2 -25346.806} C_VEL
LIN {X 0,Y 158.397,Z 365.19,A -85,B 0,C 180,E1 -25347.863,E2 -25347.863} C_VEL
LIN {X 0,Y 155.335,Z 361.375,A -85,B 0,C 180,E1 -25350.153,E2 -25350.153} C_VEL
LIN {X 0,Y 151.914,Z 357.844,A -85,B 0,C 180,E1 -25352.612,E2 -25352.612} C_VEL
LIN {X 0,Y 149.907,Z 354.669,A -85,B 0,C 180,E1 -25354.443,E2 -25354.443} C_VEL
LIN {X 0,Y 149.447,Z 353.408,A -85,B 0,C 180,E1 -25355.029,E2 -25355.029} C_VEL
LIN {X 0,Y 147.048,Z 346.385,A -85,B 0,C 180,E1 -25358.257,E2 -25358.257} C_VEL
LIN {X 0,Y 144.095,Z 338.536,A -85,B 0,C 180,E1 -25362.249,E2 -25362.249} C_VEL
LIN {X 0,Y 141.608,Z 332.993,A -85,B 0,C 180,E1 -25365.537,E2 -25365.537} C_VEL
LIN {X 0,Y 139.637,Z 328.747,A -85,B 0,C 180,E1 -25368.383,E2 -25368.383} C_VEL
LIN {X 0,Y 139.054,Z 327.557,A -85,B 0,C 180,E1 -25369.233,E2 -25369.233} C_VEL
LIN {X 0,Y 136.92,Z 323.528,A -85,B 0,C 180,E1 -25372.439,E2 -25372.439} C_VEL
LIN {X 0,Y 136.351,Z 322.045,A -85,B 0,C 180,E1 -25373.523,E2 -25373.523} C_VEL
LIN {X 0,Y 133.982,Z 319.595,A -85,B 0,C 180,E1 -25377.246,E2 -25377.246} C_VEL
LIN {X 0,Y 132.849,Z 316.513,A -85,B 0,C 180,E1 -25379.997,E2 -25379.997} C_VEL
LIN {X 0,Y 129.41,Z 314.295,A -85,B 0,C 180,E1 -25388.586,E2 -25388.586} C_VEL
LIN {X 0,Y 128.679,Z 313.236,A -85,B 0,C 180,E1 -25392.615,E2 -25392.615} C_VEL
LIN {X 0,Y 128.36,Z 313.102,A -85,B 0,C 180,E1 -25399.175,E2 -25399.175} C_VEL
LIN {X 0,Y 128.656,Z 313.968,A -85,B 0,C 180,E1 -25403.096,E2 -25403.096} C_VEL
LIN {X 0,Y 132.04,Z 316.928,A -85,B 0,C 180,E1 -25414.028,E2 -25414.028} C_VEL
LIN {X 0,Y 133.234,Z 319.847,A -85,B 0,C 180,E1 -25417.161,E2 -25417.161} C_VEL
LIN {X 0,Y 135.709,Z 322.295,A -85,B 0,C 180,E1 -25421.273,E2 -25421.273} C_VEL
LIN {X 0,Y 137.646,Z 325.857,A -85,B 0,C 180,E1 -25424.594,E2 -25424.594} C_VEL
LIN {X 0,Y 139.055,Z 327.485,A -85,B 0,C 180,E1 -25426.427,E2 -25426.427} C_VEL
LIN {X 0,Y 141.444,Z 331.329,A -85,B 0,C 180,E1 -25429.762,E2 -25429.762} C_VEL
LIN {X 0,Y 145.605,Z 338.996,A -85,B 0,C 180,E1 -25435.133,E2 -25435.133} C_VEL
LIN {X 0,Y 149.318,Z 346.549,A -85,B 0,C 180,E1 -25439.67,E2 -25439.67} C_VEL
LIN {X 0,Y 153.161,Z 355.992,A -85,B 0,C 180,E1 -25444.65,E2 -25444.65} C_VEL
LIN {X 0,Y 156.085,Z 364.878,A -85,B 0,C 180,E1 -25448.885,E2 -25448.885} C_VEL
LIN {X 0,Y 157.57,Z 370.313,A -85,B 0,C 180,E1 -25451.365,E2 -25451.365} C_VEL
LIN {X 0,Y 158.166,Z 375.98,A -85,B 0,C 180,E1 -25453.648,E2 -25453.648} C_VEL
LIN {X 0,Y 157.826,Z 377.381,A -85,B 0,C 180,E1 -25454.057,E2 -25454.057} C_VEL
LIN {X 0,Y 151.611,Z 389.84,A -85,B 0,C 180,E1 -25457.234,E2 -25457.234} C_VEL
LIN {X 0,Y 145.301,Z 401.148,A -85,B 0,C 180,E1 -25460.954,E2 -25460.954} C_VEL
LIN {X 0,Y 139.595,Z 410.567,A -85,B 0,C 180,E1 -25464.943,E2 -25464.943} C_VEL
LIN {X 0,Y 134.423,Z 418.592,A -85,B 0,C 180,E1 -25469.249,E2 -25469.249} C_VEL
LIN {X 0,Y 129.426,Z 426.39,A -85,B 0,C 180,E1 -25474.67,E2 -25474.67} C_VEL
LIN {X 0,Y 125.843,Z 431.99,A -85,B 0,C 180,E1 -25479.643,E2 -25479.643} C_VEL
LIN {X 0,Y 123.348,Z 436.184,A -85,B 0,C 180,E1 -25484.411,E2 -25484.411} C_VEL
LIN {X 0,Y 121.087,Z 440.286,A -85,B 0,C 180,E1 -25490.377,E2 -25490.377} C_VEL
LIN {X 0,Y 120.129,Z 442.299,A -85,B 0,C 180,E1 -25494.172,E2 -25494.172} C_VEL
LIN {X 0,Y 119.549,Z 443.972,A -85,B 0,C 180,E1 -25498.147,E2 -25498.147} C_VEL
LIN {X 0,Y 119.363,Z 445.839,A -85,B 0,C 180,E1 -25504.489,E2 -25504.489} C_VEL
LIN {X 0,Y 120.087,Z 446.651,A -85,B 0,C 180,E1 -25510.47,E2 -25510.47} C_VEL
LIN {X 0,Y 122.474,Z 446.443,A -85,B 0,C 180,E1 -25518.24,E2 -25518.24} C_VEL
LIN {X 0,Y 124.438,Z 445.733,A -85,B 0,C 180,E1 -25522.246,E2 -25522.246} C_VEL
LIN {X 0,Y 127.081,Z 444.494,A -85,B 0,C 180,E1 -25526.429,E2 -25526.429} C_VEL
LIN {X 0,Y 130.926,Z 442.327,A -85,B 0,C 180,E1 -25531.115,E2 -25531.115} C_VEL
LIN {X 0,Y 137.325,Z 438.257,A -85,B 0,C 180,E1 -25537.096,E2 -25537.096} C_VEL
LIN {X 0,Y 143.934,Z 433.565,A -85,B 0,C 180,E1 -25541.83,E2 -25541.83} C_VEL
LIN {X 0,Y 152.416,Z 426.782,A -85,B 0,C 180,E1 -25546.673,E2 -25546.673} C_VEL
LIN {X 0,Y 161,Z 419.142,A -85,B 0,C 180,E1 -25550.592,E2 -25550.592} C_VEL
LIN {X 0,Y 169.621,Z 410.466,A -85,B 0,C 180,E1 -25553.918,E2 -25553.918} C_VEL
LIN {X 0,Y 178.957,Z 399.78,A -85,B 0,C 180,E1 -25556.943,E2 -25556.943} C_VEL
LIN {X 0,Y 179.952,Z 397.988,A -85,B 0,C 180,E1 -25557.764,E2 -25557.764} C_VEL
LIN {X 0,Y 180.806,Z 393.879,A -85,B 0,C 180,E1 -25561.116,E2 -25561.116} C_VEL
LIN {X 0,Y 181.248,Z 390.776,A -85,B 0,C 180,E1 -25564.45,E2 -25564.45} C_VEL
LIN {X 0,Y 181.22,Z 389.328,A -85,B 0,C 180,E1 -25566.683,E2 -25566.683} C_VEL
LIN {X 0,Y 181.145,Z 387.663,A -85,B 0,C 180,E1 -25571.188,E2 -25571.188} C_VEL
LIN {X 0,Y 180.482,Z 388.4,A -85,B 0,C 180,E1 -25575.82,E2 -25575.82} C_VEL
LIN {X 0,Y 180.305,Z 389.235,A -85,B 0,C 180,E1 -25578.172,E2 -25578.172} C_VEL
LIN {X 0,Y 180.049,Z 390.683,A -85,B 0,C 180,E1 -25580.569,E2 -25580.569} C_VEL
LIN {X 0,Y 179.813,Z 392.54,A -85,B 0,C 180,E1 -25583.01,E2 -25583.01} C_VEL
LIN {X 0,Y 179.162,Z 396.687,A -85,B 0,C 180,E1 -25586.816,E2 -25586.816} C_VEL
LIN {X 0,Y 178.375,Z 400.898,A -85,B 0,C 180,E1 -25589.914,E2 -25589.914} C_VEL
LIN {X 0,Y 177.748,Z 402.755,A -85,B 0,C 180,E1 -25590.934,E2 -25590.934} C_VEL
LIN {X 0,Y 173.792,Z 410.082,A -85,B 0,C 180,E1 -25594.009,E2 -25594.009} C_VEL
LIN {X 0,Y 171.05,Z 414.515,A -85,B 0,C 180,E1 -25595.763,E2 -25595.763} C_VEL
LIN {X 0,Y 168.653,Z 417.37,A -85,B 0,C 180,E1 -25596.665,E2 -25596.665} C_VEL
LIN {X 0,Y 161.135,Z 425.385,A -85,B 0,C 180,E1 -25599.272,E2 -25599.272} C_VEL
LIN {X 0,Y 151.791,Z 434.441,A -85,B 0,C 180,E1 -25603.181,E2 -25603.181} C_VEL
LIN {X 0,Y 144.392,Z 441.071,A -85,B 0,C 180,E1 -25607.048,E2 -25607.048} C_VEL
LIN {X 0,Y 137.029,Z 447.27,A -85,B 0,C 180,E1 -25612.017,E2 -25612.017} C_VEL
LIN {X 0,Y 130.681,Z 452.224,A -85,B 0,C 180,E1 -25617.469,E2 -25617.469} C_VEL
LIN {X 0,Y 125.401,Z 456.177,A -85,B 0,C 180,E1 -25623.735,E2 -25623.735} C_VEL
LIN {X 0,Y 122.16,Z 458.713,A -85,B 0,C 180,E1 -25629.809,E2 -25629.809} C_VEL
LIN {X 0,Y 120.148,Z 460.281,A -85,B 0,C 180,E1 -25636.471,E2 -25636.471} C_VEL
LIN {X 0,Y 119.565,Z 460.765,A -85,B 0,C 180,E1 -25643.251,E2 -25643.251} C_VEL
LIN {X 0,Y 119.728,Z 460.601,A -85,B 0,C 180,E1 -25646.637,E2 -25646.637} C_VEL
LIN {X 0,Y 119.89,Z 460.137,A -85,B 0,C 180,E1 -25650.002,E2 -25650.002} C_VEL
LIN {X 0,Y 119.792,Z 459.1,A -85,B 0,C 180,E1 -25654.123,E2 -25654.123} C_VEL
LIN {X 0,Y 119.818,Z 456.769,A -85,B 0,C 180,E1 -25660.137,E2 -25660.137} C_VEL
LIN {X 0,Y 121.096,Z 452.872,A -85,B 0,C 180,E1 -25666.871,E2 -25666.871} C_VEL
LIN {X 0,Y 123.723,Z 447.591,A -85,B 0,C 180,E1 -25673.433,E2 -25673.433} C_VEL
LIN {X 0,Y 127.787,Z 440.811,A -85,B 0,C 180,E1 -25679.671,E2 -25679.671} C_VEL
LIN {X 0,Y 133.236,Z 432.357,A -85,B 0,C 180,E1 -25685.469,E2 -25685.469} C_VEL
LIN {X 0,Y 138.815,Z 423.268,A -85,B 0,C 180,E1 -25690.207,E2 -25690.207} C_VEL
LIN {X 0,Y 145.515,Z 412.419,A -85,B 0,C 180,E1 -25694.455,E2 -25694.455} C_VEL
LIN {X 0,Y 151.115,Z 402.175,A -85,B 0,C 180,E1 -25697.59,E2 -25697.59} C_VEL
LIN {X 0,Y 153.001,Z 391.17,A -85,B 0,C 180,E1 -25701.344,E2 -25701.344} C_VEL
LIN {X 0,Y 154.062,Z 379.159,A -85,B 0,C 180,E1 -25705.2,E2 -25705.2} C_VEL
LIN {X 0,Y 154.129,Z 371.564,A -85,B 0,C 180,E1 -25707.6,E2 -25707.6} C_VEL
LIN {X 0,Y 152.095,Z 362.579,A -85,B 0,C 180,E1 -25711.124,E2 -25711.124} C_VEL
LIN {X 0,Y 149.447,Z 353.408,A -85,B 0,C 180,E1 -25715.029,E2 -25715.029} C_VEL
LIN {X 0,Y 147.818,Z 350.147,A -85,B 0,C 180,E1 -25716.817,E2 -25716.817} C_VEL
LIN {X 0,Y 145.582,Z 347.771,A -85,B 0,C 180,E1 -25718.764,E2 -25718.764} C_VEL
LIN {X 0,Y 140.9,Z 343.784,A -85,B 0,C 180,E1 -25722.913,E2 -25722.913} C_VEL
LIN {X 0,Y 139.14,Z 341.146,A -85,B 0,C 180,E1 -25724.996,E2 -25724.996} C_VEL
LIN {X 0,Y 138.728,Z 340.049,A -85,B 0,C 180,E1 -25725.664,E2 -25725.664} C_VEL
LIN {X 0,Y 136.005,Z 333.597,A -85,B 0,C 180,E1 -25730.141,E2 -25730.141} C_VEL
LIN {X 0,Y 134.088,Z 329.42,A -85,B 0,C 180,E1 -25733.59,E2 -25733.59} C_VEL
LIN {X 0,Y 133.623,Z 328.39,A -85,B 0,C 180,E1 -25734.538,E2 -25734.538} C_VEL
LIN {X 0,Y 131.345,Z 325.48,A -85,B 0,C 180,E1 -25738.655,E2 -25738.655} C_VEL
LIN {X 0,Y 130.666,Z 323.238,A -85,B 0,C 180,E1 -25740.728,E2 -25740.728} C_VEL
LIN {X 0,Y 127.599,Z 321.06,A -85,B 0,C 180,E1 -25749.107,E2 -25749.107} C_VEL
LIN {X 0,Y 126.986,Z 320.128,A -85,B 0,C 180,E1 -25752.786,E2 -25752.786} C_VEL
LIN {X 0,Y 126.674,Z 320.014,A -85,B 0,C 180,E1 -25759.44,E2 -25759.44} C_VEL
LIN {X 0,Y 129.743,Z 323.449,A -85,B 0,C 180,E1 -25773.211,E2 -25773.211} C_VEL
LIN {X 0,Y 130.777,Z 326.363,A -85,B 0,C 180,E1 -25776.561,E2 -25776.561} C_VEL
LIN {X 0,Y 132.393,Z 328.146,A -85,B 0,C 180,E1 -25779.565,E2 -25779.565} C_VEL
LIN {X 0,Y 133.947,Z 331.011,A -85,B 0,C 180,E1 -25782.727,E2 -25782.727} C_VEL
LIN {X 0,Y 135.45,Z 333.014,A -85,B 0,C 180,E1 -25785.086,E2 -25785.086} C_VEL
LIN {X 0,Y 138.324,Z 338.197,A -85,B 0,C 180,E1 -25789.646,E2 -25789.646} C_VEL
LIN {X 0,Y 140.811,Z 342.883,A -85,B 0,C 180,E1 -25793.204,E2 -25793.204} C_VEL
LIN {X 0,Y 144.219,Z 350.326,A -85,B 0,C 180,E1 -25798.101,E2 -25798.101} C_VEL
LIN {X 0,Y 147.405,Z 358.395,A -85,B 0,C 180,E1 -25802.739,E2 -25802.739} C_VEL
LIN {X 0,Y 150.081,Z 366.936,A -85,B 0,C 180,E1 -25807.12,E2 -25807.12} C_VEL
LIN {X 0,Y 151.861,Z 373.834,A -85,B 0,C 180,E1 -25810.513,E2 -25810.513} C_VEL
LIN {X 0,Y 152.173,Z 376.874,A -85,B 0,C 180,E1 -25811.867,E2 -25811.867} C_VEL
LIN {X 0,Y 151.984,Z 378.818,A -85,B 0,C 180,E1 -25812.573,E2 -25812.573} C_VEL
LIN {X 0,Y 145.765,Z 390.698,A -85,B 0,C 180,E1 -25815.692,E2 -25815.692} C_VEL
LIN {X 0,Y 139.801,Z 400.944,A -85,B 0,C 180,E1 -25819.132,E2 -25819.132} C_VEL
LIN {X 0,Y 134.032,Z 410.133,A -85,B 0,C 180,E1 -25823.055,E2 -25823.055} C_VEL
LIN {X 0,Y 127.804,Z 419.371,A -85,B 0,C 180,E1 -25828.139,E2 -25828.139} C_VEL
LIN {X 0,Y 122.316,Z 427.48,A -85,B 0,C 180,E1 -25834.116,E2 -25834.116} C_VEL
LIN {X 0,Y 118.167,Z 433.744,A -85,B 0,C 180,E1 -25840.276,E2 -25840.276} C_VEL
LIN {X 0,Y 115.441,Z 438.174,A -85,B 0,C 180,E1 -25845.962,E2 -25845.962} C_VEL
LIN {X 0,Y 113.531,Z 441.616,A -85,B 0,C 180,E1 -25851.801,E2 -25851.801} C_VEL
LIN {X 0,Y 112.37,Z 444.586,A -85,B 0,C 180,E1 -25858.892,E2 -25858.892} C_VEL
LIN {X 0,Y 112.344,Z 446.364,A -85,B 0,C 180,E1 -25865.592,E2 -25865.592} C_VEL
LIN {X 0,Y 113.517,Z 447.218,A -85,B 0,C 180,E1 -25872.92,E2 -25872.92} C_VEL
LIN {X 0,Y 115.076,Z 447.104,A -85,B 0,C 180,E1 -25877.8,E2 -25877.8} C_VEL
LIN {X 0,Y 119.165,Z 445.775,A -85,B 0,C 180,E1 -25885.653,E2 -25885.653} C_VEL
LIN {X 0,Y 122.114,Z 444.433,A -85,B 0,C 180,E1 -25889.683,E2 -25889.683} C_VEL
LIN {X 0,Y 127.531,Z 441.583,A -85,B 0,C 180,E1 -25895.401,E2 -25895.401} C_VEL
LIN {X 0,Y 134.048,Z 437.596,A -85,B 0,C 180,E1 -25900.68,E2 -25900.68} C_VEL
LIN {X 0,Y 141.966,Z 432.149,A -85,B 0,C 180,E1 -25905.672,E2 -25905.672} C_VEL
LIN {X 0,Y 151.4,Z 424.803,A -85,B 0,C 180,E1 -25910.391,E2 -25910.391} C_VEL
LIN {X 0,Y 160.718,Z 416.541,A -85,B 0,C 180,E1 -25914.152,E2 -25914.152} C_VEL
LIN {X 0,Y 168.908,Z 408.364,A -85,B 0,C 180,E1 -25916.934,E2 -25916.934} C_VEL
LIN {X 0,Y 174.274,Z 402.506,A -85,B 0,C 180,E1 -25918.526,E2 -25918.526} C_VEL
LIN {X 0,Y 174.835,Z 401.742,A -85,B 0,C 180,E1 -25918.851,E2 -25918.851} C_VEL
LIN {X 0,Y 175.904,Z 397.933,A -85,B 0,C 180,E1 -25922.292,E2 -25922.292} C_VEL
LIN {X 0,Y 176.358,Z 395.688,A -85,B 0,C 180,E1 -25924.973,E2 -25924.973} C_VEL
LIN {X 0,Y 176.444,Z 394.582,A -85,B 0,C 180,E1 -25926.865,E2 -25926.865} C_VEL
LIN {X 0,Y 176.491,Z 393.103,A -85,B 0,C 180,E1 -25931.487,E2 -25931.487} C_VEL
LIN {X 0,Y 175.8,Z 394.05,A -85,B 0,C 180,E1 -25936.378,E2 -25936.378} C_VEL
LIN {X 0,Y 175.54,Z 394.991,A -85,B 0,C 180,E1 -25938.683,E2 -25938.683} C_VEL
LIN {X 0,Y 175.025,Z 397.587,A -85,B 0,C 180,E1 -25942.554,E2 -25942.554} C_VEL
LIN {X 0,Y 174.116,Z 401.561,A -85,B 0,C 180,E1 -25946.362,E2 -25946.362} C_VEL
LIN {X 0,Y 173.101,Z 405.169,A -85,B 0,C 180,E1 -25949.16,E2 -25949.16} C_VEL
LIN {X 0,Y 171.508,Z 408.205,A -85,B 0,C 180,E1 -25950.627,E2 -25950.627} C_VEL
LIN {X 0,Y 167.254,Z 414.771,A -85,B 0,C 180,E1 -25953.491,E2 -25953.491} C_VEL
LIN {X 0,Y 165.668,Z 416.855,A -85,B 0,C 180,E1 -25954.305,E2 -25954.305} C_VEL
LIN {X 0,Y 156.749,Z 425.944,A -85,B 0,C 180,E1 -25957.269,E2 -25957.269} C_VEL
LIN {X 0,Y 148.208,Z 433.789,A -85,B 0,C 180,E1 -25960.652,E2 -25960.652} C_VEL
LIN {X 0,Y 139.239,Z 441.259,A -85,B 0,C 180,E1 -25965.041,E2 -25965.041} C_VEL
LIN {X 0,Y 131.475,Z 447.359,A -85,B 0,C 180,E1 -25970.102,E2 -25970.102} C_VEL
LIN {X 0,Y 124.698,Z 452.164,A -85,B 0,C 180,E1 -25975.698,E2 -25975.698} C_VEL
LIN {X 0,Y 118.756,Z 456.164,A -85,B 0,C 180,E1 -25982.593,E2 -25982.593} C_VEL
LIN {X 0,Y 115.449,Z 458.4,A -85,B 0,C 180,E1 -25988.579,E2 -25988.579} C_VEL
LIN {X 0,Y 113.192,Z 459.912,A -85,B 0,C 180,E1 -25995.622,E2 -25995.622} C_VEL
LIN {X 0,Y 112.478,Z 460.293,A -85,B 0,C 180,E1 -26002.824,E2 -26002.824} C_VEL
LIN {X 0,Y 112.673,Z 460.083,A -85,B 0,C 180,E1 -26006.426,E2 -26006.426} C_VEL
LIN {X 0,Y 112.812,Z 459.567,A -85,B 0,C 180,E1 -26010.002,E2 -26010.002} C_VEL
LIN {X 0,Y 112.726,Z 458.6,A -85,B 0,C 180,E1 -26013.979,E2 -26013.979} C_VEL
LIN {X 0,Y 112.804,Z 456.045,A -85,B 0,C 180,E1 -26020.775,E2 -26020.775} C_VEL
LIN {X 0,Y 114.25,Z 452.072,A -85,B 0,C 180,E1 -26027.915,E2 -26027.915} C_VEL
LIN {X 0,Y 117.169,Z 446.686,A -85,B 0,C 180,E1 -26034.829,E2 -26034.829} C_VEL
LIN {X 0,Y 121.589,Z 439.78,A -85,B 0,C 180,E1 -26041.349,E2 -26041.349} C_VEL
LIN {X 0,Y 126.646,Z 432.323,A -85,B 0,C 180,E1 -26046.626,E2 -26046.626} C_VEL
LIN {X 0,Y 132.468,Z 423.319,A -85,B 0,C 180,E1 -26051.545,E2 -26051.545} C_VEL
LIN {X 0,Y 139.422,Z 412.569,A -85,B 0,C 180,E1 -26055.918,E2 -26055.918} C_VEL
LIN {X 0,Y 145.144,Z 402.405,A -85,B 0,C 180,E1 -26059.166,E2 -26059.166} C_VEL
LIN {X 0,Y 147.039,Z 392.382,A -85,B 0,C 180,E1 -26062.806,E2 -26062.806} C_VEL
LIN {X 0,Y 148.318,Z 381.299,A -85,B 0,C 180,E1 -26066.573,E2 -26066.573} C_VEL
LIN {X 0,Y 148.606,Z 375.029,A -85,B 0,C 180,E1 -26068.65,E2 -26068.65} C_VEL
LIN {X 0,Y 146.584,Z 365.011,A -85,B 0,C 180,E1 -26072.901,E2 -26072.901} C_VEL
LIN {X 0,Y 143.727,Z 354.303,A -85,B 0,C 180,E1 -26077.803,E2 -26077.803} C_VEL
LIN {X 0,Y 140.702,Z 345.292,A -85,B 0,C 180,E1 -26082.558,E2 -26082.558} C_VEL
LIN {X 0,Y 138.728,Z 340.049,A -85,B 0,C 180,E1 -26085.664,E2 -26085.664} C_VEL
LIN {X 0,Y 137.845,Z 338.109,A -85,B 0,C 180,E1 -26087.025,E2 -26087.025} C_VEL
LIN {X 0,Y 136.019,Z 336.26,A -85,B 0,C 180,E1 -26089.245,E2 -26089.245} C_VEL
LIN {X 0,Y 132.596,Z 334.823,A -85,B 0,C 180,E1 -26093.232,E2 -26093.232} C_VEL
LIN {X 0,Y 129.674,Z 333.312,A -85,B 0,C 180,E1 -26097.452,E2 -26097.452} C_VEL
LIN {X 0,Y 129.251,Z 332.775,A -85,B 0,C 180,E1 -26098.301,E2 -26098.301} C_VEL
LIN {X 0,Y 128.241,Z 329.87,A -85,B 0,C 180,E1 -26101.487,E2 -26101.487} C_VEL
LIN {X 0,Y 125.022,Z 326.947,A -85,B 0,C 180,E1 -26112.991,E2 -26112.991} C_VEL
LIN {X 0,Y 124.713,Z 326.89,A -85,B 0,C 180,E1 -26119.758,E2 -26119.758} C_VEL
LIN {X 0,Y 126.307,Z 329.484,A -85,B 0,C 180,E1 -26130.047,E2 -26130.047} C_VEL
LIN {X 0,Y 127.424,Z 330.883,A -85,B 0,C 180,E1 -26133.468,E2 -26133.468} C_VEL
LIN {X 0,Y 129.127,Z 334.127,A -85,B 0,C 180,E1 -26138.22,E2 -26138.22} C_VEL
LIN {X 0,Y 130.479,Z 336.251,A -85,B 0,C 180,E1 -26141.052,E2 -26141.052} C_VEL
LIN {X 0,Y 132.446,Z 339.693,A -85,B 0,C 180,E1 -26144.942,E2 -26144.942} C_VEL
LIN {X 0,Y 135.014,Z 344.816,A -85,B 0,C 180,E1 -26149.554,E2 -26149.554} C_VEL
LIN {X 0,Y 137.226,Z 349.429,A -85,B 0,C 180,E1 -26153.171,E2 -26153.171} C_VEL
LIN {X 0,Y 140.323,Z 357.086,A -85,B 0,C 180,E1 -26158.361,E2 -26158.361} C_VEL
LIN {X 0,Y 143.047,Z 365.192,A -85,B 0,C 180,E1 -26163.159,E2 -26163.159} C_VEL
LIN {X 0,Y 145.484,Z 374.321,A -85,B 0,C 180,E1 -26168.096,E2 -26168.096} C_VEL
LIN {X 0,Y 146.236,Z 378.787,A -85,B 0,C 180,E1 -26170.339,E2 -26170.339} C_VEL
LIN {X 0,Y 146.067,Z 380.552,A -85,B 0,C 180,E1 -26171.046,E2 -26171.046} C_VEL
LIN {X 0,Y 140.096,Z 391.43,A -85,B 0,C 180,E1 -26173.982,E2 -26173.982} C_VEL
LIN {X 0,Y 133.367,Z 402.495,A -85,B 0,C 180,E1 -26177.829,E2 -26177.829} C_VEL
LIN {X 0,Y 126.665,Z 412.506,A -85,B 0,C 180,E1 -26182.382,E2 -26182.382} C_VEL
LIN {X 0,Y 120.485,Z 421.216,A -85,B 0,C 180,E1 -26187.626,E2 -26187.626} C_VEL
LIN {X 0,Y 115.228,Z 428.546,A -85,B 0,C 180,E1 -26193.494,E2 -26193.494} C_VEL
LIN {X 0,Y 111.509,Z 433.87,A -85,B 0,C 180,E1 -26199.063,E2 -26199.063} C_VEL
LIN {X 0,Y 108.609,Z 438.328,A -85,B 0,C 180,E1 -26204.998,E2 -26204.998} C_VEL
LIN {X 0,Y 106.269,Z 442.318,A -85,B 0,C 180,E1 -26212.212,E2 -26212.212} C_VEL
LIN {X 0,Y 105.205,Z 445.186,A -85,B 0,C 180,E1 -26219.732,E2 -26219.732} C_VEL
LIN {X 0,Y 105.352,Z 446.896,A -85,B 0,C 180,E1 -26226.894,E2 -26226.894} C_VEL
LIN {X 0,Y 106.527,Z 447.634,A -85,B 0,C 180,E1 -26233.479,E2 -26233.479} C_VEL
LIN {X 0,Y 109.037,Z 447.466,A -85,B 0,C 180,E1 -26240.662,E2 -26240.662} C_VEL
LIN {X 0,Y 111.654,Z 446.763,A -85,B 0,C 180,E1 -26245.499,E2 -26245.499} C_VEL
LIN {X 0,Y 117.816,Z 444.279,A -85,B 0,C 180,E1 -26253.475,E2 -26253.475} C_VEL
LIN {X 0,Y 125.448,Z 440.353,A -85,B 0,C 180,E1 -26260.362,E2 -26260.362} C_VEL
LIN {X 0,Y 133.969,Z 435.211,A -85,B 0,C 180,E1 -26266.034,E2 -26266.034} C_VEL
LIN {X 0,Y 142.509,Z 429.291,A -85,B 0,C 180,E1 -26270.501,E2 -26270.501} C_VEL
LIN {X 0,Y 150.621,Z 423.027,A -85,B 0,C 180,E1 -26273.944,E2 -26273.944} C_VEL
LIN {X 0,Y 160.504,Z 414.355,A -85,B 0,C 180,E1 -26277.493,E2 -26277.493} C_VEL
LIN {X 0,Y 168.866,Z 406.064,A -85,B 0,C 180,E1 -26280.003,E2 -26280.003} C_VEL
LIN {X 0,Y 170.14,Z 404.121,A -85,B 0,C 180,E1 -26281.186,E2 -26281.186} C_VEL
LIN {X 0,Y 170.61,Z 402.956,A -85,B 0,C 180,E1 -26282.363,E2 -26282.363} C_VEL
LIN {X 0,Y 171.172,Z 401.034,A -85,B 0,C 180,E1 -26284.713,E2 -26284.713} C_VEL
LIN {X 0,Y 171.504,Z 399.634,A -85,B 0,C 180,E1 -26287.064,E2 -26287.064} C_VEL
LIN {X 0,Y 171.616,Z 398.524,A -85,B 0,C 180,E1 -26290.639,E2 -26290.639} C_VEL
LIN {X 0,Y 171.619,Z 398.381,A -85,B 0,C 180,E1 -26291.818,E2 -26291.818} C_VEL
LIN {X 0,Y 171.218,Z 398.732,A -85,B 0,C 180,E1 -26294.26,E2 -26294.26} C_VEL
LIN {X 0,Y 170.908,Z 399.46,A -85,B 0,C 180,E1 -26296.732,E2 -26296.732} C_VEL
LIN {X 0,Y 170.502,Z 400.642,A -85,B 0,C 180,E1 -26299.256,E2 -26299.256} C_VEL
LIN {X 0,Y 170.095,Z 402.286,A -85,B 0,C 180,E1 -26301.833,E2 -26301.833} C_VEL
LIN {X 0,Y 169.312,Z 404.764,A -85,B 0,C 180,E1 -26304.528,E2 -26304.528} C_VEL
LIN {X 0,Y 168.234,Z 407.998,A -85,B 0,C 180,E1 -26307.359,E2 -26307.359} C_VEL
LIN {X 0,Y 167.659,Z 409.307,A -85,B 0,C 180,E1 -26308.327,E2 -26308.327} C_VEL
LIN {X 0,Y 164.898,Z 413.521,A -85,B 0,C 180,E1 -26310.342,E2 -26310.342} C_VEL
LIN {X 0,Y 161.513,Z 417.983,A -85,B 0,C 180,E1 -26312.31,E2 -26312.31} C_VEL
LIN {X 0,Y 151.28,Z 427.715,A -85,B 0,C 180,E1 -26315.614,E2 -26315.614} C_VEL
LIN {X 0,Y 141.236,Z 436.165,A -85,B 0,C 180,E1 -26319.533,E2 -26319.533} C_VEL
LIN {X 0,Y 132.122,Z 443.079,A -85,B 0,C 180,E1 -26324.105,E2 -26324.105} C_VEL
LIN {X 0,Y 124.118,Z 448.665,A -85,B 0,C 180,E1 -26329.373,E2 -26329.373} C_VEL
LIN {X 0,Y 118.827,Z 452.12,A -85,B 0,C 180,E1 -26333.743,E2 -26333.743} C_VEL
LIN {X 0,Y 112.14,Z 456.176,A -85,B 0,C 180,E1 -26341.337,E2 -26341.337} C_VEL
LIN {X 0,Y 108.784,Z 458.09,A -85,B 0,C 180,E1 -26347.196,E2 -26347.196} C_VEL
LIN {X 0,Y 106.274,Z 459.505,A -85,B 0,C 180,E1 -26354.664,E2 -26354.664} C_VEL
LIN {X 0,Y 105.421,Z 459.818,A -85,B 0,C 180,E1 -26362.341,E2 -26362.341} C_VEL
LIN {X 0,Y 105.617,Z 459.524,A -85,B 0,C 180,E1 -26366.555,E2 -26366.555} C_VEL
LIN {X 0,Y 105.737,Z 458.992,A -85,B 0,C 180,E1 -26370.003,E2 -26370.003} C_VEL
LIN {X 0,Y 105.66,Z 458.094,A -85,B 0,C 180,E1 -26373.816,E2 -26373.816} C_VEL
LIN {X 0,Y 105.789,Z 455.308,A -85,B 0,C 180,E1 -26381.499,E2 -26381.499} C_VEL
LIN {X 0,Y 107.447,Z 451.224,A -85,B 0,C 180,E1 -26389.092,E2 -26389.092} C_VEL
LIN {X 0,Y 110.666,Z 445.729,A -85,B 0,C 180,E1 -26396.397,E2 -26396.397} C_VEL
LIN {X 0,Y 115.495,Z 438.693,A -85,B 0,C 180,E1 -26403.209,E2 -26403.209} C_VEL
LIN {X 0,Y 120.95,Z 431.152,A -85,B 0,C 180,E1 -26408.659,E2 -26408.659} C_VEL
LIN {X 0,Y 126.94,Z 422.303,A -85,B 0,C 180,E1 -26413.55,E2 -26413.55} C_VEL
LIN {X 0,Y 134.508,Z 411.047,A -85,B 0,C 180,E1 -26418.124,E2 -26418.124} C_VEL
LIN {X 0,Y 138.931,Z 403.689,A -85,B 0,C 180,E1 -26420.486,E2 -26420.486} C_VEL
LIN {X 0,Y 141.032,Z 394.311,A -85,B 0,C 180,E1 -26424.077,E2 -26424.077} C_VEL
LIN {X 0,Y 142.483,Z 384.408,A -85,B 0,C 180,E1 -26427.641,E2 -26427.641} C_VEL
LIN {X 0,Y 142.969,Z 377.881,A -85,B 0,C 180,E1 -26429.985,E2 -26429.985} C_VEL
LIN {X 0,Y 141.66,Z 370.154,A -85,B 0,C 180,E1 -26433.477,E2 -26433.477} C_VEL
LIN {X 0,Y 139.671,Z 361.144,A -85,B 0,C 180,E1 -26437.825,E2 -26437.825} C_VEL
LIN {X 0,Y 137.833,Z 354.357,A -85,B 0,C 180,E1 -26441.414,E2 -26441.414} C_VEL
LIN {X 0,Y 135.911,Z 348.268,A -85,B 0,C 180,E1 -26445.013,E2 -26445.013} C_VEL
LIN {X 0,Y 134.391,Z 343.897,A -85,B 0,C 180,E1 -26447.923,E2 -26447.923} C_VEL
LIN {X 0,Y 132.906,Z 339.751,A -85,B 0,C 180,E1 -26450.869,E2 -26450.869} C_VEL
LIN {X 0,Y 130.808,Z 334.699,A -85,B 0,C 180,E1 -26455.367,E2 -26455.367} C_VEL
LIN {X 0,Y 129.251,Z 332.775,A -85,B 0,C 180,E1 -26458.301,E2 -26458.301} C_VEL
LIN {X 0,Y 127.983,Z 331.835,A -85,B 0,C 180,E1 -26460.828,E2 -26460.828} C_VEL
LIN {X 0,Y 126.51,Z 332.058,A -85,B 0,C 180,E1 -26463.419,E2 -26463.419} C_VEL
LIN {X 0,Y 123.841,Z 333.708,A -85,B 0,C 180,E1 -26468.76,E2 -26468.76} C_VEL
LIN {X 0,Y 123.006,Z 333.978,A -85,B 0,C 180,E1 -26471.531,E2 -26471.531} C_VEL
LIN {X 0,Y 122.867,Z 333.839,A -85,B 0,C 180,E1 -26472.463,E2 -26472.463} C_VEL
LIN {X 0,Y 122.531,Z 333.534,A -85,B 0,C 180,E1 -26476.662,E2 -26476.662} C_VEL
LIN {X 0,Y 122.489,Z 333.687,A -85,B 0,C 180,E1 -26480.133,E2 -26480.133} C_VEL
LIN {X 0,Y 124.021,Z 336.456,A -85,B 0,C 180,E1 -26490.66,E2 -26490.66} C_VEL
LIN {X 0,Y 124.477,Z 337.023,A -85,B 0,C 180,E1 -26492.119,E2 -26492.119} C_VEL
LIN {X 0,Y 126.744,Z 341.338,A -85,B 0,C 180,E1 -26499.074,E2 -26499.074} C_VEL
LIN {X 0,Y 129.285,Z 346.499,A -85,B 0,C 180,E1 -26505.031,E2 -26505.031} C_VEL
LIN {X 0,Y 131.087,Z 350.315,A -85,B 0,C 180,E1 -26508.635,E2 -26508.635} C_VEL
LIN {X 0,Y 133.622,Z 356.522,A -85,B 0,C 180,E1 -26513.655,E2 -26513.655} C_VEL
LIN {X 0,Y 135.816,Z 362.631,A -85,B 0,C 180,E1 -26517.952,E2 -26517.952} C_VEL
LIN {X 0,Y 138.035,Z 370.234,A -85,B 0,C 180,E1 -26522.725,E2 -26522.725} C_VEL
LIN {X 0,Y 139.778,Z 377.858,A -85,B 0,C 180,E1 -26527.152,E2 -26527.152} C_VEL
LIN {X 0,Y 140.321,Z 380.847,A -85,B 0,C 180,E1 -26528.793,E2 -26528.793} C_VEL
LIN {X 0,Y 140.144,Z 382.322,A -85,B 0,C 180,E1 -26529.447,E2 -26529.447} C_VEL
LIN {X 0,Y 133.242,Z 394.173,A -85,B 0,C 180,E1 -26532.819,E2 -26532.819} C_VEL
LIN {X 0,Y 126.973,Z 403.905,A -85,B 0,C 180,E1 -26536.392,E2 -26536.392} C_VEL
LIN {X 0,Y 120.603,Z 412.992,A -85,B 0,C 180,E1 -26540.691,E2 -26540.691} C_VEL
LIN {X 0,Y 113.744,Z 422.161,A -85,B 0,C 180,E1 -26546.455,E2 -26546.455} C_VEL
LIN {X 0,Y 108.89,Z 428.568,A -85,B 0,C 180,E1 -26551.847,E2 -26551.847} C_VEL
LIN {X 0,Y 104.883,Z 433.981,A -85,B 0,C 180,E1 -26557.699,E2 -26557.699} C_VEL
LIN {X 0,Y 101.589,Z 438.776,A -85,B 0,C 180,E1 -26564.433,E2 -26564.433} C_VEL
LIN {X 0,Y 99.021,Z 443.022,A -85,B 0,C 180,E1 -26572.693,E2 -26572.693} C_VEL
LIN {X 0,Y 98.059,Z 445.782,A -85,B 0,C 180,E1 -26580.687,E2 -26580.687} C_VEL
LIN {X 0,Y 98.603,Z 447.647,A -85,B 0,C 180,E1 -26589.898,E2 -26589.898} C_VEL
LIN {X 0,Y 99.834,Z 448.124,A -85,B 0,C 180,E1 -26595.26,E2 -26595.26} C_VEL
LIN {X 0,Y 103.645,Z 447.778,A -85,B 0,C 180,E1 -26604.454,E2 -26604.454} C_VEL
LIN {X 0,Y 106.524,Z 446.976,A -85,B 0,C 180,E1 -26609.052,E2 -26609.052} C_VEL
LIN {X 0,Y 110.077,Z 445.713,A -85,B 0,C 180,E1 -26613.458,E2 -26613.458} C_VEL
LIN {X 0,Y 115.126,Z 443.552,A -85,B 0,C 180,E1 -26618.518,E2 -26618.518} C_VEL
LIN {X 0,Y 123.686,Z 439.235,A -85,B 0,C 180,E1 -26624.999,E2 -26624.999} C_VEL
LIN {X 0,Y 131.726,Z 434.542,A -85,B 0,C 180,E1 -26629.67,E2 -26629.67} C_VEL
LIN {X 0,Y 141.824,Z 427.773,A -85,B 0,C 180,E1 -26634.315,E2 -26634.315} C_VEL
LIN {X 0,Y 151.854,Z 420.021,A -85,B 0,C 180,E1 -26638.015,E2 -26638.015} C_VEL
LIN {X 0,Y 161.665,Z 411.371,A -85,B 0,C 180,E1 -26641.033,E2 -26641.033} C_VEL
LIN {X 0,Y 164.205,Z 408.907,A -85,B 0,C 180,E1 -26641.736,E2 -26641.736} C_VEL
LIN {X 0,Y 165.078,Z 407.819,A -85,B 0,C 180,E1 -26642.443,E2 -26642.443} C_VEL
LIN {X 0,Y 165.841,Z 405.899,A -85,B 0,C 180,E1 -26644.865,E2 -26644.865} C_VEL
LIN {X 0,Y 166.369,Z 404.517,A -85,B 0,C 180,E1 -26647.283,E2 -26647.283} C_VEL
LIN {X 0,Y 166.525,Z 403.752,A -85,B 0,C 180,E1 -26649.721,E2 -26649.721} C_VEL
LIN {X 0,Y 166.524,Z 403.467,A -85,B 0,C 180,E1 -26652.185,E2 -26652.185} C_VEL
LIN {X 0,Y 166.116,Z 403.909,A -85,B 0,C 180,E1 -26654.708,E2 -26654.708} C_VEL
LIN {X 0,Y 165.746,Z 404.753,A -85,B 0,C 180,E1 -26657.269,E2 -26657.269} C_VEL
LIN {X 0,Y 165.095,Z 406.496,A -85,B 0,C 180,E1 -26660.529,E2 -26660.529} C_VEL
LIN {X 0,Y 164.531,Z 408.024,A -85,B 0,C 180,E1 -26662.611,E2 -26662.611} C_VEL
LIN {X 0,Y 162.98,Z 411.871,A -85,B 0,C 180,E1 -26666.403,E2 -26666.403} C_VEL
LIN {X 0,Y 162.081,Z 413.355,A -85,B 0,C 180,E1 -26667.427,E2 -26667.427} C_VEL
LIN {X 0,Y 158.657,Z 417.71,A -85,B 0,C 180,E1 -26669.546,E2 -26669.546} C_VEL
LIN {X 0,Y 157.252,Z 419.32,A -85,B 0,C 180,E1 -26670.296,E2 -26670.296} C_VEL
LIN {X 0,Y 147.278,Z 428.289,A -85,B 0,C 180,E1 -26673.379,E2 -26673.379} C_VEL
LIN {X 0,Y 136.821,Z 436.518,A -85,B 0,C 180,E1 -26677.237,E2 -26677.237} C_VEL
LIN {X 0,Y 126.542,Z 443.752,A -85,B 0,C 180,E1 -26682.189,E2 -26682.189} C_VEL
LIN {X 0,Y 118.781,Z 448.728,A -85,B 0,C 180,E1 -26687.126,E2 -26687.126} C_VEL
LIN {X 0,Y 113.122,Z 452.044,A -85,B 0,C 180,E1 -26691.594,E2 -26691.594} C_VEL
LIN {X 0,Y 106.826,Z 455.47,A -85,B 0,C 180,E1 -26698.247,E2 -26698.247} C_VEL
LIN {X 0,Y 102.194,Z 457.79,A -85,B 0,C 180,E1 -26705.633,E2 -26705.633} C_VEL
LIN {X 0,Y 99.379,Z 459.083,A -85,B 0,C 180,E1 -26713.571,E2 -26713.571} C_VEL
LIN {X 0,Y 98.345,Z 459.337,A -85,B 0,C 180,E1 -26721.786,E2 -26721.786} C_VEL
LIN {X 0,Y 98.535,Z 458.908,A -85,B 0,C 180,E1 -26726.981,E2 -26726.981} C_VEL
LIN {X 0,Y 98.665,Z 458.41,A -85,B 0,C 180,E1 -26730.003,E2 -26730.003} C_VEL
LIN {X 0,Y 98.563,Z 457.452,A -85,B 0,C 180,E1 -26734.092,E2 -26734.092} C_VEL
LIN {X 0,Y 98.807,Z 454.548,A -85,B 0,C 180,E1 -26742.324,E2 -26742.324} C_VEL
LIN {X 0,Y 100.698,Z 450.338,A -85,B 0,C 180,E1 -26750.427,E2 -26750.427} C_VEL
LIN {X 0,Y 104.271,Z 444.709,A -85,B 0,C 180,E1 -26758.155,E2 -26758.155} C_VEL
LIN {X 0,Y 109.536,Z 437.529,A -85,B 0,C 180,E1 -26765.275,E2 -26765.275} C_VEL
LIN {X 0,Y 115.396,Z 429.838,A -85,B 0,C 180,E1 -26770.901,E2 -26770.901} C_VEL
LIN {X 0,Y 121.297,Z 421.599,A -85,B 0,C 180,E1 -26775.53,E2 -26775.53} C_VEL
LIN {X 0,Y 128.676,Z 411.118,A -85,B 0,C 180,E1 -26779.879,E2 -26779.879} C_VEL
LIN {X 0,Y 133.117,Z 403.762,A -85,B 0,C 180,E1 -26782.37,E2 -26782.37} C_VEL
LIN {X 0,Y 135.393,Z 394.375,A -85,B 0,C 180,E1 -26786.157,E2 -26786.157} C_VEL
LIN {X 0,Y 137.083,Z 384.282,A -85,B 0,C 180,E1 -26790.006,E2 -26790.006} C_VEL
LIN {X 0,Y 137.35,Z 380.372,A -85,B 0,C 180,E1 -26791.56,E2 -26791.56} C_VEL
LIN {X 0,Y 135.847,Z 370.601,A -85,B 0,C 180,E1 -26796.36,E2 -26796.36} C_VEL
LIN {X 0,Y 134.12,Z 361.967,A -85,B 0,C 180,E1 -26800.946,E2 -26800.946} C_VEL
LIN {X 0,Y 132.258,Z 354.583,A -85,B 0,C 180,E1 -26805.377,E2 -26805.377} C_VEL
LIN {X 0,Y 130.589,Z 349.209,A -85,B 0,C 180,E1 -26809.14,E2 -26809.14} C_VEL
LIN {X 0,Y 129.329,Z 345.224,A -85,B 0,C 180,E1 -26812.189,E2 -26812.189} C_VEL
LIN {X 0,Y 128.107,Z 341.908,A -85,B 0,C 180,E1 -26815.269,E2 -26815.269} C_VEL
LIN {X 0,Y 127.429,Z 340.511,A -85,B 0,C 180,E1 -26816.835,E2 -26816.835} C_VEL
LIN {X 0,Y 125.869,Z 337.54,A -85,B 0,C 180,E1 -26820.946,E2 -26820.946} C_VEL
LIN {X 0,Y 125.115,Z 336.241,A -85,B 0,C 180,E1 -26823.217,E2 -26823.217} C_VEL
LIN {X 0,Y 122.867,Z 333.839,A -85,B 0,C 180,E1 -26832.463,E2 -26832.463} C_VEL
LIN {X 0,Y 122.594,Z 333.841,A -85,B 0,C 180,E1 -26834.287,E2 -26834.287} C_VEL
LIN {X 0,Y 121.979,Z 335.038,A -85,B 0,C 180,E1 -26836.986,E2 -26836.986} C_VEL
LIN {X 0,Y 120.457,Z 340.053,A -85,B 0,C 180,E1 -26843.184,E2 -26843.184} C_VEL
LIN {X 0,Y 120.36,Z 341.69,A -85,B 0,C 180,E1 -26845.959,E2 -26845.959} C_VEL
LIN {X 0,Y 120.462,Z 341.992,A -85,B 0,C 180,E1 -26846.907,E2 -26846.907} C_VEL
LIN {X 0,Y 121.498,Z 343.304,A -85,B 0,C 180,E1 -26851.368,E2 -26851.368} C_VEL
LIN {X 0,Y 123.524,Z 347.72,A -85,B 0,C 180,E1 -26858.74,E2 -26858.74} C_VEL
LIN {X 0,Y 125.139,Z 351.205,A -85,B 0,C 180,E1 -26863.102,E2 -26863.102} C_VEL
LIN {X 0,Y 127.358,Z 356.605,A -85,B 0,C 180,E1 -26868.53,E2 -26868.53} C_VEL
LIN {X 0,Y 129.784,Z 363.574,A -85,B 0,C 180,E1 -26874.312,E2 -26874.312} C_VEL
LIN {X 0,Y 131.554,Z 369.779,A -85,B 0,C 180,E1 -26878.727,E2 -26878.727} C_VEL
LIN {X 0,Y 132.99,Z 375.656,A -85,B 0,C 180,E1 -26882.602,E2 -26882.602} C_VEL
LIN {X 0,Y 134.422,Z 383.555,A -85,B 0,C 180,E1 -26887.47,E2 -26887.47} C_VEL
LIN {X 0,Y 133.096,Z 386.318,A -85,B 0,C 180,E1 -26888.305,E2 -26888.305} C_VEL
LIN {X 0,Y 125.595,Z 398.259,A -85,B 0,C 180,E1 -26892.028,E2 -26892.028} C_VEL
LIN {X 0,Y 118.396,Z 408.495,A -85,B 0,C 180,E1 -26896.262,E2 -26896.262} C_VEL
LIN {X 0,Y 110.782,Z 418.415,A -85,B 0,C 180,E1 -26901.791,E2 -26901.791} C_VEL
LIN {X 0,Y 104.281,Z 426.642,A -85,B 0,C 180,E1 -26908.147,E2 -26908.147} C_VEL
LIN {X 0,Y 98.814,Z 433.473,A -85,B 0,C 180,E1 -26915.351,E2 -26915.351} C_VEL
LIN {X 0,Y 94.324,Z 439.542,A -85,B 0,C 180,E1 -26924.412,E2 -26924.412} C_VEL
LIN {X 0,Y 91.768,Z 443.669,A -85,B 0,C 180,E1 -26933.231,E2 -26933.231} C_VEL
LIN {X 0,Y 90.914,Z 446.617,A -85,B 0,C 180,E1 -26942.757,E2 -26942.757} C_VEL
LIN {X 0,Y 91.478,Z 447.912,A -85,B 0,C 180,E1 -26949.809,E2 -26949.809} C_VEL
LIN {X 0,Y 93.68,Z 448.624,A -85,B 0,C 180,E1 -26958.604,E2 -26958.604} C_VEL
LIN {X 0,Y 96.103,Z 448.464,A -85,B 0,C 180,E1 -26964.2,E2 -26964.2} C_VEL
LIN {X 0,Y 102.199,Z 447.006,A -85,B 0,C 180,E1 -26973.371,E2 -26973.371} C_VEL
LIN {X 0,Y 106.286,Z 445.61,A -85,B 0,C 180,E1 -26977.77,E2 -26977.77} C_VEL
LIN {X 0,Y 113.416,Z 442.659,A -85,B 0,C 180,E1 -26983.83,E2 -26983.83} C_VEL
LIN {X 0,Y 121.658,Z 438.665,A -85,B 0,C 180,E1 -26989.118,E2 -26989.118} C_VEL
LIN {X 0,Y 130.992,Z 433.325,A -85,B 0,C 180,E1 -26993.843,E2 -26993.843} C_VEL
LIN {X 0,Y 142.309,Z 425.851,A -85,B 0,C 180,E1 -26998.298,E2 -26998.298} C_VEL
LIN {X 0,Y 152.92,Z 417.64,A -85,B 0,C 180,E1 -27001.695,E2 -27001.695} C_VEL
LIN {X 0,Y 157.986,Z 413.259,A -85,B 0,C 180,E1 -27003.11,E2 -27003.11} C_VEL
LIN {X 0,Y 159.855,Z 411.462,A -85,B 0,C 180,E1 -27003.784,E2 -27003.784} C_VEL
LIN {X 0,Y 160.333,Z 410.576,A -85,B 0,C 180,E1 -27005.032,E2 -27005.032} C_VEL
LIN {X 0,Y 161.051,Z 409.217,A -85,B 0,C 180,E1 -27007.525,E2 -27007.525} C_VEL
LIN {X 0,Y 161.283,Z 408.51,A -85,B 0,C 180,E1 -27010.041,E2 -27010.041} C_VEL
LIN {X 0,Y 161.227,Z 408.36,A -85,B 0,C 180,E1 -27012.591,E2 -27012.591} C_VEL
LIN {X 0,Y 160.683,Z 409.108,A -85,B 0,C 180,E1 -27015.801,E2 -27015.801} C_VEL
LIN {X 0,Y 160.272,Z 409.935,A -85,B 0,C 180,E1 -27017.878,E2 -27017.878} C_VEL
LIN {X 0,Y 159.197,Z 412.42,A -85,B 0,C 180,E1 -27022.022,E2 -27022.022} C_VEL
LIN {X 0,Y 157.646,Z 415.49,A -85,B 0,C 180,E1 -27025.333,E2 -27025.333} C_VEL
LIN {X 0,Y 156.677,Z 416.848,A -85,B 0,C 180,E1 -27026.221,E2 -27026.221} C_VEL
LIN {X 0,Y 153.378,Z 420.474,A -85,B 0,C 180,E1 -27028.061,E2 -27028.061} C_VEL
LIN {X 0,Y 143.5,Z 428.836,A -85,B 0,C 180,E1 -27031.015,E2 -27031.015} C_VEL
LIN {X 0,Y 132.65,Z 436.876,A -85,B 0,C 180,E1 -27034.798,E2 -27034.798} C_VEL
LIN {X 0,Y 123.04,Z 443.216,A -85,B 0,C 180,E1 -27039.101,E2 -27039.101} C_VEL
LIN {X 0,Y 113.647,Z 448.787,A -85,B 0,C 180,E1 -27044.674,E2 -27044.674} C_VEL
LIN {X 0,Y 107.6,Z 451.965,A -85,B 0,C 180,E1 -27049.223,E2 -27049.223} C_VEL
LIN {X 0,Y 100.794,Z 455.294,A -85,B 0,C 180,E1 -27056.099,E2 -27056.099} C_VEL
LIN {X 0,Y 95.691,Z 457.494,A -85,B 0,C 180,E1 -27063.857,E2 -27063.857} C_VEL
LIN {X 0,Y 92.514,Z 458.662,A -85,B 0,C 180,E1 -27072.313,E2 -27072.313} C_VEL
LIN {X 0,Y 91.291,Z 458.806,A -85,B 0,C 180,E1 -27081.146,E2 -27081.146} C_VEL
LIN {X 0,Y 91.471,Z 458.236,A -85,B 0,C 180,E1 -27087.304,E2 -27087.304} C_VEL
LIN {X 0,Y 91.58,Z 457.826,A -85,B 0,C 180,E1 -27090.003,E2 -27090.003} C_VEL
LIN {X 0,Y 91.478,Z 456.813,A -85,B 0,C 180,E1 -27094.409,E2 -27094.409} C_VEL
LIN {X 0,Y 91.825,Z 453.788,A -85,B 0,C 180,E1 -27103.277,E2 -27103.277} C_VEL
LIN {X 0,Y 94.017,Z 449.455,A -85,B 0,C 180,E1 -27111.951,E2 -27111.951} C_VEL
LIN {X 0,Y 97.993,Z 443.691,A -85,B 0,C 180,E1 -27120.138,E2 -27120.138} C_VEL
LIN {X 0,Y 103.748,Z 436.37,A -85,B 0,C 180,E1 -27127.569,E2 -27127.569} C_VEL
LIN {X 0,Y 110.021,Z 428.511,A -85,B 0,C 180,E1 -27133.372,E2 -27133.372} C_VEL
LIN {X 0,Y 116.138,Z 420.462,A -85,B 0,C 180,E1 -27137.899,E2 -27137.899} C_VEL
LIN {X 0,Y 122.963,Z 411.16,A -85,B 0,C 180,E1 -27141.806,E2 -27141.806} C_VEL
LIN {X 0,Y 127.061,Z 404.899,A -85,B 0,C 180,E1 -27143.996,E2 -27143.996} C_VEL
LIN {X 0,Y 129.396,Z 396.693,A -85,B 0,C 180,E1 -27147.472,E2 -27147.472} C_VEL
LIN {X 0,Y 131.318,Z 387.485,A -85,B 0,C 180,E1 -27151.202,E2 -27151.202} C_VEL
LIN {X 0,Y 131.713,Z 385.067,A -85,B 0,C 180,E1 -27152.164,E2 -27152.164} C_VEL
LIN {X 0,Y 131.431,Z 380.055,A -85,B 0,C 180,E1 -27154.67,E2 -27154.67} C_VEL
LIN {X 0,Y 130.186,Z 371.013,A -85,B 0,C 180,E1 -27159.592,E2 -27159.592} C_VEL
LIN {X 0,Y 128.815,Z 363.303,A -85,B 0,C 180,E1 -27164.166,E2 -27164.166} C_VEL
LIN {X 0,Y 127.478,Z 357.569,A -85,B 0,C 180,E1 -27168.065,E2 -27168.065} C_VEL
LIN {X 0,Y 126.113,Z 352.482,A -85,B 0,C 180,E1 -27171.988,E2 -27171.988} C_VEL
LIN {X 0,Y 125.109,Z 348.952,A -85,B 0,C 180,E1 -27175.155,E2 -27175.155} C_VEL
LIN {X 0,Y 124.565,Z 347.359,A -85,B 0,C 180,E1 -27176.762,E2 -27176.762} C_VEL
LIN {X 0,Y 122.975,Z 343.862,A -85,B 0,C 180,E1 -27181.634,E2 -27181.634} C_VEL
LIN {X 0,Y 122.489,Z 342.918,A -85,B 0,C 180,E1 -27183.286,E2 -27183.286} C_VEL
LIN {X 0,Y 120.301,Z 340.32,A -85,B 0,C 180,E1 -27193.51,E2 -27193.51} C_VEL
LIN {X 0,Y 120.056,Z 340.195,A -85,B 0,C 180,E1 -27197.016,E2 -27197.016} C_VEL
LIN {X 0,Y 119.965,Z 340.49,A -85,B 0,C 180,E1 -27200.575,E2 -27200.575} C_VEL
LIN {X 0,Y 120.462,Z 341.992,A -85,B 0,C 180,E1 -27206.907,E2 -27206.907} C_VEL
LIN {X 0,Y 120.699,Z 342.791,A -85,B 0,C 180,E1 -27208.73,E2 -27208.73} C_VEL
LIN {X 0,Y 120.76,Z 344.168,A -85,B 0,C 180,E1 -27210.48,E2 -27210.48} C_VEL
LIN {X 0,Y 120.513,Z 347.948,A -85,B 0,C 180,E1 -27213.802,E2 -27213.802} C_VEL
LIN {X 0,Y 120.328,Z 354.057,A -85,B 0,C 180,E1 -27218.814,E2 -27218.814} C_VEL
LIN {X 0,Y 120.731,Z 355.597,A -85,B 0,C 180,E1 -27220.578,E2 -27220.578} C_VEL
LIN {X 0,Y 122.229,Z 359.472,A -85,B 0,C 180,E1 -27225.19,E2 -27225.19} C_VEL
LIN {X 0,Y 124.007,Z 364.804,A -85,B 0,C 180,E1 -27230.313,E2 -27230.313} C_VEL
LIN {X 0,Y 125.472,Z 369.884,A -85,B 0,C 180,E1 -27234.571,E2 -27234.571} C_VEL
LIN {X 0,Y 127.173,Z 377.48,A -85,B 0,C 180,E1 -27240.171,E2 -27240.171} C_VEL
LIN {X 0,Y 128.358,Z 385.079,A -85,B 0,C 180,E1 -27245.263,E2 -27245.263} C_VEL
LIN {X 0,Y 128.331,Z 386.388,A -85,B 0,C 180,E1 -27245.994,E2 -27245.994} C_VEL
LIN {X 0,Y 120.804,Z 397.932,A -85,B 0,C 180,E1 -27249.568,E2 -27249.568} C_VEL
LIN {X 0,Y 113.312,Z 408.184,A -85,B 0,C 180,E1 -27253.791,E2 -27253.791} C_VEL
LIN {X 0,Y 105.25,Z 418.237,A -85,B 0,C 180,E1 -27259.416,E2 -27259.416} C_VEL
LIN {X 0,Y 98.361,Z 426.482,A -85,B 0,C 180,E1 -27265.9,E2 -27265.9} C_VEL
LIN {X 0,Y 93.273,Z 432.373,A -85,B 0,C 180,E1 -27272.156,E2 -27272.156} C_VEL
LIN {X 0,Y 89.321,Z 437.31,A -85,B 0,C 180,E1 -27279.051,E2 -27279.051} C_VEL
LIN {X 0,Y 86.326,Z 441.342,A -85,B 0,C 180,E1 -27286.554,E2 -27286.554} C_VEL
LIN {X 0,Y 84.392,Z 444.542,A -85,B 0,C 180,E1 -27294.603,E2 -27294.603} C_VEL
LIN {X 0,Y 83.828,Z 446.931,A -85,B 0,C 180,E1 -27303.041,E2 -27303.041} C_VEL
LIN {X 0,Y 84.645,Z 448.419,A -85,B 0,C 180,E1 -27311.655,E2 -27311.655} C_VEL
LIN {X 0,Y 86.794,Z 449.094,A -85,B 0,C 180,E1 -27319.632,E2 -27319.632} C_VEL
LIN {X 0,Y 90.889,Z 448.828,A -85,B 0,C 180,E1 -27328.268,E2 -27328.268} C_VEL
LIN {X 0,Y 94.512,Z 448.119,A -85,B 0,C 180,E1 -27333.507,E2 -27333.507} C_VEL
LIN {X 0,Y 99.848,Z 446.609,A -85,B 0,C 180,E1 -27339.399,E2 -27339.399} C_VEL
LIN {X 0,Y 108.437,Z 443.466,A -85,B 0,C 180,E1 -27346.442,E2 -27346.442} C_VEL
LIN {X 0,Y 117.108,Z 439.575,A -85,B 0,C 180,E1 -27351.722,E2 -27351.722} C_VEL
LIN {X 0,Y 128.046,Z 433.768,A -85,B 0,C 180,E1 -27356.857,E2 -27356.857} C_VEL
LIN {X 0,Y 138.199,Z 427.415,A -85,B 0,C 180,E1 -27360.579,E2 -27360.579} C_VEL
LIN {X 0,Y 149.709,Z 419.046,A -85,B 0,C 180,E1 -27364.026,E2 -27364.026} C_VEL
LIN {X 0,Y 154.284,Z 415.325,A -85,B 0,C 180,E1 -27365.23,E2 -27365.23} C_VEL
LIN {X 0,Y 155.561,Z 413.72,A -85,B 0,C 180,E1 -27367.792,E2 -27367.792} C_VEL
LIN {X 0,Y 155.847,Z 413.074,A -85,B 0,C 180,E1 -27370.395,E2 -27370.395} C_VEL
LIN {X 0,Y 155.714,Z 413.085,A -85,B 0,C 180,E1 -27373.045,E2 -27373.045} C_VEL
LIN {X 0,Y 155.222,Z 413.761,A -85,B 0,C 180,E1 -27375.766,E2 -27375.766} C_VEL
LIN {X 0,Y 154.519,Z 414.966,A -85,B 0,C 180,E1 -27378.568,E2 -27378.568} C_VEL
LIN {X 0,Y 153.678,Z 416.677,A -85,B 0,C 180,E1 -27381.463,E2 -27381.463} C_VEL
LIN {X 0,Y 152.832,Z 418.034,A -85,B 0,C 180,E1 -27383.122,E2 -27383.122} C_VEL
LIN {X 0,Y 151.667,Z 419.651,A -85,B 0,C 180,E1 -27384.651,E2 -27384.651} C_VEL
LIN {X 0,Y 148.722,Z 422.586,A -85,B 0,C 180,E1 -27386.126,E2 -27386.126} C_VEL
LIN {X 0,Y 137.125,Z 431.569,A -85,B 0,C 180,E1 -27389.395,E2 -27389.395} C_VEL
LIN {X 0,Y 126.012,Z 439.009,A -85,B 0,C 180,E1 -27393.223,E2 -27393.223} C_VEL
LIN {X 0,Y 115.745,Z 445.083,A -85,B 0,C 180,E1 -27397.879,E2 -27397.879} C_VEL
LIN {X 0,Y 106.481,Z 449.907,A -85,B 0,C 180,E1 -27403.45,E2 -27403.45} C_VEL
LIN {X 0,Y 98.434,Z 453.617,A -85,B 0,C 180,E1 -27410.019,E2 -27410.019} C_VEL
LIN {X 0,Y 91.882,Z 456.279,A -85,B 0,C 180,E1 -27417.631,E2 -27417.631} C_VEL
LIN {X 0,Y 87.246,Z 457.852,A -85,B 0,C 180,E1 -27426.252,E2 -27426.252} C_VEL
LIN {X 0,Y 84.735,Z 458.386,A -85,B 0,C 180,E1 -27435.596,E2 -27435.596} C_VEL
LIN {X 0,Y 84.283,Z 457.884,A -85,B 0,C 180,E1 -27445.22,E2 -27445.22} C_VEL
LIN {X 0,Y 84.52,Z 457.207,A -85,B 0,C 180,E1 -27450.003,E2 -27450.003} C_VEL
LIN {X 0,Y 84.377,Z 456.15,A -85,B 0,C 180,E1 -27454.781,E2 -27454.781} C_VEL
LIN {X 0,Y 84.889,Z 453.003,A -85,B 0,C 180,E1 -27464.385,E2 -27464.385} C_VEL
LIN {X 0,Y 87.411,Z 448.539,A -85,B 0,C 180,E1 -27473.707,E2 -27473.707} C_VEL
LIN {X 0,Y 92.393,Z 441.993,A -85,B 0,C 180,E1 -27483.196,E2 -27483.196} C_VEL
LIN {X 0,Y 99.08,Z 434.152,A -85,B 0,C 180,E1 -27491.009,E2 -27491.009} C_VEL
LIN {X 0,Y 105.916,Z 425.889,A -85,B 0,C 180,E1 -27496.881,E2 -27496.881} C_VEL
LIN {X 0,Y 113.545,Z 416.286,A -85,B 0,C 180,E1 -27501.829,E2 -27501.829} C_VEL
LIN {X 0,Y 121.115,Z 405.852,A -85,B 0,C 180,E1 -27505.784,E2 -27505.784} C_VEL
LIN {X 0,Y 123.33,Z 399.27,A -85,B 0,C 180,E1 -27508.74,E2 -27508.74} C_VEL
LIN {X 0,Y 125.541,Z 390.585,A -85,B 0,C 180,E1 -27512.492,E2 -27512.492} C_VEL
LIN {X 0,Y 126.127,Z 387.143,A -85,B 0,C 180,E1 -27514.023,E2 -27514.023} C_VEL
LIN {X 0,Y 125.728,Z 380.314,A -85,B 0,C 180,E1 -27517.829,E2 -27517.829} C_VEL
LIN {X 0,Y 124.768,Z 371.288,A -85,B 0,C 180,E1 -27523.26,E2 -27523.26} C_VEL
LIN {X 0,Y 123.49,Z 363.623,A -85,B 0,C 180,E1 -27528.507,E2 -27528.507} C_VEL
LIN {X 0,Y 122.232,Z 357.611,A -85,B 0,C 180,E1 -27533.393,E2 -27533.393} C_VEL
LIN {X 0,Y 121.368,Z 354.177,A -85,B 0,C 180,E1 -27536.677,E2 -27536.677} C_VEL
LIN {X 0,Y 119.98,Z 350.545,A -85,B 0,C 180,E1 -27541.675,E2 -27541.675} C_VEL
LIN {X 0,Y 119.592,Z 349.488,A -85,B 0,C 180,E1 -27543.365,E2 -27543.365} C_VEL
LIN {X 0,Y 117.954,Z 347.548,A -85,B 0,C 180,E1 -27550.293,E2 -27550.293} C_VEL
LIN {X 0,Y 117.55,Z 346.849,A -85,B 0,C 180,E1 -27553.832,E2 -27553.832} C_VEL
LIN {X 0,Y 117.309,Z 346.779,A -85,B 0,C 180,E1 -27557.427,E2 -27557.427} C_VEL
LIN {X 0,Y 117.182,Z 347.182,A -85,B 0,C 180,E1 -27561.087,E2 -27561.087} C_VEL
LIN {X 0,Y 117.866,Z 348.891,A -85,B 0,C 180,E1 -27568.486,E2 -27568.486} C_VEL
LIN {X 0,Y 118.622,Z 350.322,A -85,B 0,C 180,E1 -27572.219,E2 -27572.219} C_VEL
LIN {X 0,Y 119.927,Z 353.56,A -85,B 0,C 180,E1 -27577.802,E2 -27577.802} C_VEL
LIN {X 0,Y 120.731,Z 355.597,A -85,B 0,C 180,E1 -27580.578,E2 -27580.578} C_VEL
LIN {X 0,Y 121.169,Z 357.179,A -85,B 0,C 180,E1 -27582.269,E2 -27582.269} C_VEL
LIN {X 0,Y 121.25,Z 359.233,A -85,B 0,C 180,E1 -27583.858,E2 -27583.858} C_VEL
LIN {X 0,Y 120.831,Z 364.125,A -85,B 0,C 180,E1 -27586.822,E2 -27586.822} C_VEL
LIN {X 0,Y 120.126,Z 371.711,A -85,B 0,C 180,E1 -27591.335,E2 -27591.335} C_VEL
LIN {X 0,Y 120.347,Z 373.803,A -85,B 0,C 180,E1 -27592.977,E2 -27592.977} C_VEL
LIN {X 0,Y 121.699,Z 380.929,A -85,B 0,C 180,E1 -27598.683,E2 -27598.683} C_VEL
LIN {X 0,Y 122.544,Z 387.72,A -85,B 0,C 180,E1 -27603.608,E2 -27603.608} C_VEL
LIN {X 0,Y 121.813,Z 389.461,A -85,B 0,C 180,E1 -27604.358,E2 -27604.358} C_VEL
LIN {X 0,Y 113.654,Z 401.11,A -85,B 0,C 180,E1 -27608.219,E2 -27608.219} C_VEL
LIN {X 0,Y 105.929,Z 410.962,A -85,B 0,C 180,E1 -27612.626,E2 -27612.626} C_VEL
LIN {X 0,Y 98.771,Z 419.355,A -85,B 0,C 180,E1 -27617.672,E2 -27617.672} C_VEL
LIN {X 0,Y 91.829,Z 427.176,A -85,B 0,C 180,E1 -27624.178,E2 -27624.178} C_VEL
LIN {X 0,Y 85.758,Z 433.88,A -85,B 0,C 180,E1 -27631.942,E2 -27631.942} C_VEL
LIN {X 0,Y 81.48,Z 438.844,A -85,B 0,C 180,E1 -27639.93,E2 -27639.93} C_VEL
LIN {X 0,Y 78.589,Z 442.691,A -85,B 0,C 180,E1 -27648.236,E2 -27648.236} C_VEL
LIN {X 0,Y 76.955,Z 445.672,A -85,B 0,C 180,E1 -27657.166,E2 -27657.166} C_VEL
LIN {X 0,Y 76.775,Z 447.482,A -85,B 0,C 180,E1 -27664.538,E2 -27664.538} C_VEL
LIN {X 0,Y 78.377,Z 449.163,A -85,B 0,C 180,E1 -27675.831,E2 -27675.831} C_VEL
LIN {X 0,Y 80.498,Z 449.571,A -85,B 0,C 180,E1 -27682.335,E2 -27682.335} C_VEL
LIN {X 0,Y 84.327,Z 449.398,A -85,B 0,C 180,E1 -27690.003,E2 -27690.003} C_VEL
LIN {X 0,Y 90.698,Z 448.268,A -85,B 0,C 180,E1 -27698.404,E2 -27698.404} C_VEL
LIN {X 0,Y 95.496,Z 446.988,A -85,B 0,C 180,E1 -27703.073,E2 -27703.073} C_VEL
LIN {X 0,Y 101.853,Z 444.912,A -85,B 0,C 180,E1 -27708.058,E2 -27708.058} C_VEL
LIN {X 0,Y 112.948,Z 440.458,A -85,B 0,C 180,E1 -27714.579,E2 -27714.579} C_VEL
LIN {X 0,Y 122.501,Z 435.792,A -85,B 0,C 180,E1 -27718.87,E2 -27718.87} C_VEL
LIN {X 0,Y 134.363,Z 428.984,A -85,B 0,C 180,E1 -27723.001,E2 -27723.001} C_VEL
LIN {X 0,Y 145.678,Z 421.317,A -85,B 0,C 180,E1 -27726.175,E2 -27726.175} C_VEL
LIN {X 0,Y 148.669,Z 419.092,A -85,B 0,C 180,E1 -27726.93,E2 -27726.93} C_VEL
LIN {X 0,Y 149.838,Z 418.035,A -85,B 0,C 180,E1 -27728.092,E2 -27728.092} C_VEL
LIN {X 0,Y 150.238,Z 417.445,A -85,B 0,C 180,E1 -27730.787,E2 -27730.787} C_VEL
LIN {X 0,Y 149.984,Z 417.633,A -85,B 0,C 180,E1 -27733.553,E2 -27733.553} C_VEL
LIN {X 0,Y 149.422,Z 418.428,A -85,B 0,C 180,E1 -27736.395,E2 -27736.395} C_VEL
LIN {X 0,Y 148.017,Z 420.709,A -85,B 0,C 180,E1 -27740.864,E2 -27740.864} C_VEL
LIN {X 0,Y 147.026,Z 422.017,A -85,B 0,C 180,E1 -27742.486,E2 -27742.486} C_VEL
LIN {X 0,Y 145.617,Z 423.402,A -85,B 0,C 180,E1 -27743.513,E2 -27743.513} C_VEL
LIN {X 0,Y 142.735,Z 425.731,A -85,B 0,C 180,E1 -27744.374,E2 -27744.374} C_VEL
LIN {X 0,Y 130.841,Z 434.072,A -85,B 0,C 180,E1 -27747.595,E2 -27747.595} C_VEL
LIN {X 0,Y 119.487,Z 440.938,A -85,B 0,C 180,E1 -27751.481,E2 -27751.481} C_VEL
LIN {X 0,Y 108.966,Z 446.496,A -85,B 0,C 180,E1 -27756.277,E2 -27756.277} C_VEL
LIN {X 0,Y 101.702,Z 449.94,A -85,B 0,C 180,E1 -27760.528,E2 -27760.528} C_VEL
LIN {X 0,Y 93.056,Z 453.491,A -85,B 0,C 180,E1 -27767.182,E2 -27767.182} C_VEL
LIN {X 0,Y 85.899,Z 455.996,A -85,B 0,C 180,E1 -27775.064,E2 -27775.064} C_VEL
LIN {X 0,Y 80.728,Z 457.498,A -85,B 0,C 180,E1 -27784.2,E2 -27784.2} C_VEL
LIN {X 0,Y 77.822,Z 457.903,A -85,B 0,C 180,E1 -27794.284,E2 -27794.284} C_VEL
LIN {X 0,Y 77.191,Z 457.284,A -85,B 0,C 180,E1 -27804.78,E2 -27804.78} C_VEL
LIN {X 0,Y 77.443,Z 456.55,A -85,B 0,C 180,E1 -27810.004,E2 -27810.004} C_VEL
LIN {X 0,Y 77.285,Z 455.438,A -85,B 0,C 180,E1 -27815.221,E2 -27815.221} C_VEL
LIN {X 0,Y 78.002,Z 452.21,A -85,B 0,C 180,E1 -27825.686,E2 -27825.686} C_VEL
LIN {X 0,Y 80.899,Z 447.614,A -85,B 0,C 180,E1 -27835.749,E2 -27835.749} C_VEL
LIN {X 0,Y 86.092,Z 441.326,A -85,B 0,C 180,E1 -27845.273,E2 -27845.273} C_VEL
LIN {X 0,Y 92.786,Z 433.945,A -85,B 0,C 180,E1 -27852.98,E2 -27852.98} C_VEL
LIN {X 0,Y 100.008,Z 425.733,A -85,B 0,C 180,E1 -27859.069,E2 -27859.069} C_VEL
LIN {X 0,Y 107.084,Z 417.29,A -85,B 0,C 180,E1 -27863.616,E2 -27863.616} C_VEL
LIN {X 0,Y 114.624,Z 407.629,A -85,B 0,C 180,E1 -27867.469,E2 -27867.469} C_VEL
LIN {X 0,Y 115.801,Z 405.777,A -85,B 0,C 180,E1 -27868.179,E2 -27868.179} C_VEL
LIN {X 0,Y 118.864,Z 396.704,A -85,B 0,C 180,E1 -27872.491,E2 -27872.491} C_VEL
LIN {X 0,Y 120.449,Z 390.859,A -85,B 0,C 180,E1 -27875.145,E2 -27875.145} C_VEL
LIN {X 0,Y 120.437,Z 384.293,A -85,B 0,C 180,E1 -27879.019,E2 -27879.019} C_VEL
LIN {X 0,Y 119.902,Z 375.434,A -85,B 0,C 180,E1 -27884.703,E2 -27884.703} C_VEL
LIN {X 0,Y 119.089,Z 368.479,A -85,B 0,C 180,E1 -27889.799,E2 -27889.799} C_VEL
LIN {X 0,Y 118.201,Z 362.611,A -85,B 0,C 180,E1 -27894.88,E2 -27894.88} C_VEL
LIN {X 0,Y 117.52,Z 359.383,A -85,B 0,C 180,E1 -27898.283,E2 -27898.283} C_VEL
LIN {X 0,Y 116.418,Z 355.961,A -85,B 0,C 180,E1 -27903.457,E2 -27903.457} C_VEL
LIN {X 0,Y 114.762,Z 353.742,A -85,B 0,C 180,E1 -27911.513,E2 -27911.513} C_VEL
LIN {X 0,Y 114.52,Z 353.267,A -85,B 0,C 180,E1 -27914.206,E2 -27914.206} C_VEL
LIN {X 0,Y 114.27,Z 353.285,A -85,B 0,C 180,E1 -27917.906,E2 -27917.906} C_VEL
LIN {X 0,Y 114.323,Z 354.589,A -85,B 0,C 180,E1 -27925.484,E2 -27925.484} C_VEL
LIN {X 0,Y 115.143,Z 356.313,A -85,B 0,C 180,E1 -27931.289,E2 -27931.289} C_VEL
LIN {X 0,Y 116.489,Z 360.315,A -85,B 0,C 180,E1 -27938.339,E2 -27938.339} C_VEL
LIN {X 0,Y 118.095,Z 364.996,A -85,B 0,C 180,E1 -27944.424,E2 -27944.424} C_VEL
LIN {X 0,Y 119.54,Z 370.337,A -85,B 0,C 180,E1 -27949.838,E2 -27949.838} C_VEL
LIN {X 0,Y 120.347,Z 373.803,A -85,B 0,C 180,E1 -27952.977,E2 -27952.977} C_VEL
LIN {X 0,Y 120.304,Z 376.156,A -85,B 0,C 180,E1 -27954.491,E2 -27954.491} C_VEL
LIN {X 0,Y 118.725,Z 380.975,A -85,B 0,C 180,E1 -27956.592,E2 -27956.592} C_VEL
LIN {X 0,Y 116.921,Z 385.876,A -85,B 0,C 180,E1 -27958.727,E2 -27958.727} C_VEL
LIN {X 0,Y 116.576,Z 388.345,A -85,B 0,C 180,E1 -27960.283,E2 -27960.283} C_VEL
LIN {X 0,Y 116.677,Z 389.49,A -85,B 0,C 180,E1 -27961.189,E2 -27961.189} C_VEL
LIN {X 0,Y 116.437,Z 390.945,A -85,B 0,C 180,E1 -27962.107,E2 -27962.107} C_VEL
LIN {X 0,Y 108.512,Z 401.723,A -85,B 0,C 180,E1 -27965.717,E2 -27965.717} C_VEL
LIN {X 0,Y 99.908,Z 412.122,A -85,B 0,C 180,E1 -27970.477,E2 -27970.477} C_VEL
LIN {X 0,Y 91.248,Z 421.612,A -85,B 0,C 180,E1 -27976.637,E2 -27976.637} C_VEL
LIN {X 0,Y 84.061,Z 429.13,A -85,B 0,C 180,E1 -27983.644,E2 -27983.644} C_VEL
LIN {X 0,Y 77.406,Z 436.085,A -85,B 0,C 180,E1 -27993.009,E2 -27993.009} C_VEL
LIN {X 0,Y 73.646,Z 440.346,A -85,B 0,C 180,E1 -28000.999,E2 -28000.999} C_VEL
LIN {X 0,Y 70.875,Z 443.94,A -85,B 0,C 180,E1 -28010.303,E2 -28010.303} C_VEL
LIN {X 0,Y 69.638,Z 446.763,A -85,B 0,C 180,E1 -28020.301,E2 -28020.301} C_VEL
LIN {X 0,Y 69.812,Z 448.151,A -85,B 0,C 180,E1 -28027.154,E2 -28027.154} C_VEL
LIN {X 0,Y 71.295,Z 449.42,A -85,B 0,C 180,E1 -28036.376,E2 -28036.376} C_VEL
LIN {X 0,Y 75.215,Z 450.046,A -85,B 0,C 180,E1 -28047.233,E2 -28047.233} C_VEL
LIN {X 0,Y 78.841,Z 449.871,A -85,B 0,C 180,E1 -28053.538,E2 -28053.538} C_VEL
